(* PLC project Adressering.ecp, WAGO e!COCKPIT e!COCKPIT *)
(* stored: creationDateTime 2021-01-18T14:20:23.2110188, modificationDateTime 2021-01-18T11:51:27.6823754 *)

TYPE dtRomtype_1 : STRUCT
  RB601_V : BOOL;  (* Bevegelse *)
END_STRUCT;
END_TYPE

TYPE dtRomtype_11 : STRUCT
  RB601_V : BOOL;  (* Bevegelse *)
  RB601_HVAC : BOOL;  (* HVAC signal *)
END_STRUCT;
END_TYPE

TYPE dtRomtype_111 : STRUCT
  RB601_V : BOOL;  (* Bevegelse *)
  RB601_HVAC : BOOL;  (* HVAC signal *)
  RT601_CT : REAL;  (* Rom temperatur *)
  RT601_SP_D : REAL;  (* Temperatur SP *)
  RT601_SP_S : REAL;  (* Temperatur SP standby *)
  RT601_SP_N : REAL;  (* Temperatur SP nattsenk *)
  RT601_SP_F : REAL;  (* Temperatur SP frostsikring *)
  RT601_CS : REAL;  (* Aktivt temperatur SP *)
  OPM : REAL;  (* Rom modus *)
  OPM_CV : REAL;  (* Rom modus verdi *)
END_STRUCT;
END_TYPE

TYPE dtRomtype_1111 : STRUCT
  RB601_V : BOOL;  (* Bevegelse *)
  RB601_HVAC : BOOL;  (* HVAC signal *)
  RT601_CT : REAL;  (* Rom temperatur *)
  RT601_SP_D : REAL;  (* Temperatur SP *)
  RT601_SP_S : REAL;  (* Temperatur SP standby *)
  RT601_SP_N : REAL;  (* Temperatur SP nattsenk *)
  RT601_SP_F : REAL;  (* Temperatur SP frostsikring *)
  RT601_CS : REAL;  (* Aktivt temperatur SP *)
  OPM : REAL;  (* Rom modus *)
  OPM_CV : REAL;  (* Rom modus verdi *)
  RY601_CV : REAL;  (* Co2 Nivaa *)
  RY601_SP : REAL;  (* Co2 SP *)
  RY601_OP : REAL;  (* Co2 paadrag *)
END_STRUCT;
END_TYPE

TYPE dtRomtype_11101 : STRUCT
  RB601_V : BOOL;  (* Bevegelse *)
  RB601_HVAC : BOOL;  (* HVAC signal *)
  RT601_CT : REAL;  (* Rom temperatur *)
  RT601_SP_D : REAL;  (* Temperatur SP *)
  RT601_SP_S : REAL;  (* Temperatur SP standby *)
  RT601_SP_N : REAL;  (* Temperatur SP nattsenk *)
  RT601_SP_F : REAL;  (* Temperatur SP frostsikring *)
  RT601_CS : REAL;  (* Aktivt temperatur SP *)
  OPM : REAL;  (* Rom modus *)
  OPM_CV : REAL;  (* Rom modus verdi *)
  LH601_OP : REAL;  (* Varmepaadrag *)
  SB601_MAN : REAL;  (* Varmepaadrag force *)
END_STRUCT;
END_TYPE

TYPE dtRomtype_111011 : STRUCT
  RB601_V : BOOL;  (* Bevegelse *)
  RB601_HVAC : BOOL;  (* HVAC signal *)
  RT601_CT : REAL;  (* Rom temperatur *)
  RT601_SP_D : REAL;  (* Temperatur SP *)
  RT601_SP_S : REAL;  (* Temperatur SP standby *)
  RT601_SP_N : REAL;  (* Temperatur SP nattsenk *)
  RT601_SP_F : REAL;  (* Temperatur SP frostsikring *)
  RT601_CS : REAL;  (* Aktivt temperatur SP *)
  OPM : REAL;  (* Rom modus *)
  OPM_CV : REAL;  (* Rom modus verdi *)
  LH601_OP : REAL;  (* Varmepaadrag *)
  SB601_MAN : REAL;  (* Varmepaadrag force *)
  LH601_CMD : BOOL;  (* LH601_CMD *)
END_STRUCT;
END_TYPE

TYPE dtRomtype_1110111 : STRUCT
  RB601_V : BOOL;  (* Bevegelse *)
  RB601_HVAC : BOOL;  (* HVAC signal *)
  RT601_CT : REAL;  (* Rom temperatur *)
  RT601_SP_D : REAL;  (* Temperatur SP *)
  RT601_SP_S : REAL;  (* Temperatur SP standby *)
  RT601_SP_N : REAL;  (* Temperatur SP nattsenk *)
  RT601_SP_F : REAL;  (* Temperatur SP frostsikring *)
  RT601_CS : REAL;  (* Aktivt temperatur SP *)
  OPM : REAL;  (* Rom modus *)
  OPM_CV : REAL;  (* Rom modus verdi *)
  LH601_OP : REAL;  (* Varmepaadrag *)
  SB601_MAN : REAL;  (* Varmepaadrag force *)
  LH601_CMD : BOOL;  (* LH601_CMD *)
  LC601_OP : REAL;  (* LC601_OP *)
  LC601_MAN : REAL;  (* LC601 Force *)
END_STRUCT;
END_TYPE

TYPE dtRomtype_11111111 : STRUCT
  RB601_V : BOOL;  (* Bevegelse *)
  RB601_HVAC : BOOL;  (* HVAC signal *)
  RT601_CT : REAL;  (* Rom temperatur *)
  RT601_SP_D : REAL;  (* Temperatur SP *)
  RT601_SP_S : REAL;  (* Temperatur SP standby *)
  RT601_SP_N : REAL;  (* Temperatur SP nattsenk *)
  RT601_SP_F : REAL;  (* Temperatur SP frostsikring *)
  RT601_CS : REAL;  (* Aktivt temperatur SP *)
  OPM : REAL;  (* Rom modus *)
  OPM_CV : REAL;  (* Rom modus verdi *)
  RY601_CV : REAL;  (* Co2 Nivaa *)
  RY601_SP : REAL;  (* Co2 SP *)
  RY601_OP : REAL;  (* Co2 paadrag *)
  LH601_OP : REAL;  (* Varmepaadrag *)
  SB601_MAN : REAL;  (* Varmepaadrag force *)
  LH601_CMD : BOOL;  (* LH601_CMD *)
  LC601_OP : REAL;  (* LC601_OP *)
  LC601_MAN : REAL;  (* LC601 Force *)
  LC601_CMD : BOOL;  (* LC601_CMD *)
END_STRUCT;
END_TYPE

TYPE dtRomtype_111010111 : STRUCT
  RB601_V : BOOL;  (* Bevegelse *)
  RB601_HVAC : BOOL;  (* HVAC signal *)
  RT601_CT : REAL;  (* Rom temperatur *)
  RT601_SP_D : REAL;  (* Temperatur SP *)
  RT601_SP_S : REAL;  (* Temperatur SP standby *)
  RT601_SP_N : REAL;  (* Temperatur SP nattsenk *)
  RT601_SP_F : REAL;  (* Temperatur SP frostsikring *)
  RT601_CS : REAL;  (* Aktivt temperatur SP *)
  OPM : REAL;  (* Rom modus *)
  OPM_CV : REAL;  (* Rom modus verdi *)
  LH601_OP : REAL;  (* Varmepaadrag *)
  SB601_MAN : REAL;  (* Varmepaadrag force *)
  LC601_OP : REAL;  (* LC601_OP *)
  LC601_MAN : REAL;  (* LC601 Force *)
  LC601_CMD : BOOL;  (* LC601_CMD *)
  RT601_SP : REAL;  (* Temperatur SP feedback *)
END_STRUCT;
END_TYPE

TYPE dtRomtype_1111101011 : STRUCT
  RB601_V : BOOL;  (* Bevegelse *)
  RB601_HVAC : BOOL;  (* HVAC signal *)
  RT601_CT : REAL;  (* Rom temperatur *)
  RT601_SP_D : REAL;  (* Temperatur SP *)
  RT601_SP_S : REAL;  (* Temperatur SP standby *)
  RT601_SP_N : REAL;  (* Temperatur SP nattsenk *)
  RT601_SP_F : REAL;  (* Temperatur SP frostsikring *)
  RT601_CS : REAL;  (* Aktivt temperatur SP *)
  OPM : REAL;  (* Rom modus *)
  OPM_CV : REAL;  (* Rom modus verdi *)
  RY601_CV : REAL;  (* Co2 Nivaa *)
  RY601_SP : REAL;  (* Co2 SP *)
  RY601_OP : REAL;  (* Co2 paadrag *)
  LH601_OP : REAL;  (* Varmepaadrag *)
  SB601_MAN : REAL;  (* Varmepaadrag force *)
  LC601_OP : REAL;  (* LC601_OP *)
  LC601_MAN : REAL;  (* LC601 Force *)
  RT601_SP : REAL;  (* Temperatur SP feedback *)
  RT601_SP_FB : REAL;  (* Temperatur SP *)
  RT601_SP_IN : REAL;  (* Temperatur SP lokalt panel *)
END_STRUCT;
END_TYPE

TYPE dtRomtype_2111111111 : STRUCT
  RB601_V : BOOL;  (* Bevegelse *)
  RB602_V : BOOL;  (* Bevegelse *)
  RB601_HVAC : BOOL;  (* HVAC signal *)
  RT601_CT : REAL;  (* Rom temperatur *)
  RT601_SP_D : REAL;  (* Temperatur SP *)
  RT601_SP_S : REAL;  (* Temperatur SP standby *)
  RT601_SP_N : REAL;  (* Temperatur SP nattsenk *)
  RT601_SP_F : REAL;  (* Temperatur SP frostsikring *)
  RT601_CS : REAL;  (* Aktivt temperatur SP *)
  OPM : REAL;  (* Rom modus *)
  OPM_CV : REAL;  (* Rom modus verdi *)
  RY601_CV : REAL;  (* Co2 Nivaa *)
  RY601_SP : REAL;  (* Co2 SP *)
  RY601_OP : REAL;  (* Co2 paadrag *)
  LH601_OP : REAL;  (* Varmepaadrag *)
  SB601_MAN : REAL;  (* Varmepaadrag force *)
  LH601_CMD : BOOL;  (* LH601_CMD *)
  LC601_OP : REAL;  (* LC601_OP *)
  LC601_MAN : REAL;  (* LC601 Force *)
  LC601_CMD : BOOL;  (* LC601_CMD *)
  RT601_SP : REAL;  (* Temperatur SP feedback *)
  RT601_SP_FB : REAL;  (* Temperatur SP *)
  RT601_SP_IN : REAL;  (* Temperatur SP lokalt panel *)
END_STRUCT;
END_TYPE

TYPE dtRomtype_1211111111 : STRUCT
  RB601_V : BOOL;  (* Bevegelse *)
  RB601_HVAC : BOOL;  (* HVAC signal *)
  RB602_HVAC : BOOL;  (* HVAC signal *)
  RT601_CT : REAL;  (* Rom temperatur *)
  RT601_SP_D : REAL;  (* Temperatur SP *)
  RT601_SP_S : REAL;  (* Temperatur SP standby *)
  RT601_SP_N : REAL;  (* Temperatur SP nattsenk *)
  RT601_SP_F : REAL;  (* Temperatur SP frostsikring *)
  RT601_CS : REAL;  (* Aktivt temperatur SP *)
  OPM : REAL;  (* Rom modus *)
  OPM_CV : REAL;  (* Rom modus verdi *)
  RY601_CV : REAL;  (* Co2 Nivaa *)
  RY601_SP : REAL;  (* Co2 SP *)
  RY601_OP : REAL;  (* Co2 paadrag *)
  LH601_OP : REAL;  (* Varmepaadrag *)
  SB601_MAN : REAL;  (* Varmepaadrag force *)
  LH601_CMD : BOOL;  (* LH601_CMD *)
  LC601_OP : REAL;  (* LC601_OP *)
  LC601_MAN : REAL;  (* LC601 Force *)
  LC601_CMD : BOOL;  (* LC601_CMD *)
  RT601_SP : REAL;  (* Temperatur SP feedback *)
  RT601_SP_FB : REAL;  (* Temperatur SP *)
  RT601_SP_IN : REAL;  (* Temperatur SP lokalt panel *)
END_STRUCT;
END_TYPE

TYPE dtRomtype_1121111111 : STRUCT
  RB601_V : BOOL;  (* Bevegelse *)
  RB601_HVAC : BOOL;  (* HVAC signal *)
  RT601_CT : REAL;  (* Rom temperatur *)
  RT602_CT : REAL;  (* Rom temperatur *)
  RT601_SP_D : REAL;  (* Temperatur SP *)
  RT601_SP_S : REAL;  (* Temperatur SP standby *)
  RT601_SP_N : REAL;  (* Temperatur SP nattsenk *)
  RT601_SP_F : REAL;  (* Temperatur SP frostsikring *)
  RT601_CS : REAL;  (* Aktivt temperatur SP *)
  OPM : REAL;  (* Rom modus *)
  OPM_CV : REAL;  (* Rom modus verdi *)
  RY601_CV : REAL;  (* Co2 Nivaa *)
  RY601_SP : REAL;  (* Co2 SP *)
  RY601_OP : REAL;  (* Co2 paadrag *)
  LH601_OP : REAL;  (* Varmepaadrag *)
  SB601_MAN : REAL;  (* Varmepaadrag force *)
  LH601_CMD : BOOL;  (* LH601_CMD *)
  LC601_OP : REAL;  (* LC601_OP *)
  LC601_MAN : REAL;  (* LC601 Force *)
  LC601_CMD : BOOL;  (* LC601_CMD *)
  RT601_SP : REAL;  (* Temperatur SP feedback *)
  RT601_SP_FB : REAL;  (* Temperatur SP *)
  RT601_SP_IN : REAL;  (* Temperatur SP lokalt panel *)
END_STRUCT;
END_TYPE

TYPE dtRomtype_1112111111 : STRUCT
  RB601_V : BOOL;  (* Bevegelse *)
  RB601_HVAC : BOOL;  (* HVAC signal *)
  RT601_CT : REAL;  (* Rom temperatur *)
  RT601_SP_D : REAL;  (* Temperatur SP *)
  RT601_SP_S : REAL;  (* Temperatur SP standby *)
  RT601_SP_N : REAL;  (* Temperatur SP nattsenk *)
  RT601_SP_F : REAL;  (* Temperatur SP frostsikring *)
  RT601_CS : REAL;  (* Aktivt temperatur SP *)
  OPM : REAL;  (* Rom modus *)
  OPM_CV : REAL;  (* Rom modus verdi *)
  RY601_CV : REAL;  (* Co2 Nivaa *)
  RY601_SP : REAL;  (* Co2 SP *)
  RY601_OP : REAL;  (* Co2 paadrag *)
  RY602_CV : REAL;  (* Co2 Nivaa *)
  RY602_SP : REAL;  (* Co2 SP *)
  RY602_OP : REAL;  (* Co2 paadrag *)
  LH601_OP : REAL;  (* Varmepaadrag *)
  SB601_MAN : REAL;  (* Varmepaadrag force *)
  LH601_CMD : BOOL;  (* LH601_CMD *)
  LC601_OP : REAL;  (* LC601_OP *)
  LC601_MAN : REAL;  (* LC601 Force *)
  LC601_CMD : BOOL;  (* LC601_CMD *)
  RT601_SP : REAL;  (* Temperatur SP feedback *)
  RT601_SP_FB : REAL;  (* Temperatur SP *)
  RT601_SP_IN : REAL;  (* Temperatur SP lokalt panel *)
END_STRUCT;
END_TYPE

TYPE dtRomtype_1111211111 : STRUCT
  RB601_V : BOOL;  (* Bevegelse *)
  RB601_HVAC : BOOL;  (* HVAC signal *)
  RT601_CT : REAL;  (* Rom temperatur *)
  RT601_SP_D : REAL;  (* Temperatur SP *)
  RT601_SP_S : REAL;  (* Temperatur SP standby *)
  RT601_SP_N : REAL;  (* Temperatur SP nattsenk *)
  RT601_SP_F : REAL;  (* Temperatur SP frostsikring *)
  RT601_CS : REAL;  (* Aktivt temperatur SP *)
  OPM : REAL;  (* Rom modus *)
  OPM_CV : REAL;  (* Rom modus verdi *)
  RY601_CV : REAL;  (* Co2 Nivaa *)
  RY601_SP : REAL;  (* Co2 SP *)
  RY601_OP : REAL;  (* Co2 paadrag *)
  LH601_OP : REAL;  (* Varmepaadrag *)
  LH602_OP : REAL;  (* Varmepaadrag *)
  SB601_MAN : REAL;  (* Varmepaadrag force *)
  LH601_CMD : BOOL;  (* LH601_CMD *)
  LC601_OP : REAL;  (* LC601_OP *)
  LC601_MAN : REAL;  (* LC601 Force *)
  LC601_CMD : BOOL;  (* LC601_CMD *)
  RT601_SP : REAL;  (* Temperatur SP feedback *)
  RT601_SP_FB : REAL;  (* Temperatur SP *)
  RT601_SP_IN : REAL;  (* Temperatur SP lokalt panel *)
END_STRUCT;
END_TYPE

TYPE dtRomtype_1111112111 : STRUCT
  RB601_V : BOOL;  (* Bevegelse *)
  RB601_HVAC : BOOL;  (* HVAC signal *)
  RT601_CT : REAL;  (* Rom temperatur *)
  RT601_SP_D : REAL;  (* Temperatur SP *)
  RT601_SP_S : REAL;  (* Temperatur SP standby *)
  RT601_SP_N : REAL;  (* Temperatur SP nattsenk *)
  RT601_SP_F : REAL;  (* Temperatur SP frostsikring *)
  RT601_CS : REAL;  (* Aktivt temperatur SP *)
  OPM : REAL;  (* Rom modus *)
  OPM_CV : REAL;  (* Rom modus verdi *)
  RY601_CV : REAL;  (* Co2 Nivaa *)
  RY601_SP : REAL;  (* Co2 SP *)
  RY601_OP : REAL;  (* Co2 paadrag *)
  LH601_OP : REAL;  (* Varmepaadrag *)
  SB601_MAN : REAL;  (* Varmepaadrag force *)
  LH601_CMD : BOOL;  (* LH601_CMD *)
  LC601_OP : REAL;  (* LC601_OP *)
  LC602_OP : REAL;  (* LC602_OP *)
  LC601_MAN : REAL;  (* LC601 Force *)
  LC601_CMD : BOOL;  (* LC601_CMD *)
  RT601_SP : REAL;  (* Temperatur SP feedback *)
  RT601_SP_FB : REAL;  (* Temperatur SP *)
  RT601_SP_IN : REAL;  (* Temperatur SP lokalt panel *)
END_STRUCT;
END_TYPE

TYPE dtRomtype_1111111211 : STRUCT
  RB601_V : BOOL;  (* Bevegelse *)
  RB601_HVAC : BOOL;  (* HVAC signal *)
  RT601_CT : REAL;  (* Rom temperatur *)
  RT601_SP_D : REAL;  (* Temperatur SP *)
  RT601_SP_S : REAL;  (* Temperatur SP standby *)
  RT601_SP_N : REAL;  (* Temperatur SP nattsenk *)
  RT601_SP_F : REAL;  (* Temperatur SP frostsikring *)
  RT601_CS : REAL;  (* Aktivt temperatur SP *)
  OPM : REAL;  (* Rom modus *)
  OPM_CV : REAL;  (* Rom modus verdi *)
  RY601_CV : REAL;  (* Co2 Nivaa *)
  RY601_SP : REAL;  (* Co2 SP *)
  RY601_OP : REAL;  (* Co2 paadrag *)
  LH601_OP : REAL;  (* Varmepaadrag *)
  SB601_MAN : REAL;  (* Varmepaadrag force *)
  LH601_CMD : BOOL;  (* LH601_CMD *)
  LC601_OP : REAL;  (* LC601_OP *)
  LC601_MAN : REAL;  (* LC601 Force *)
  LC601_CMD : BOOL;  (* LC601_CMD *)
  LC602_CMD : BOOL;  (* LC602_CMD *)
  RT601_SP : REAL;  (* Temperatur SP feedback *)
  RT601_SP_FB : REAL;  (* Temperatur SP *)
  RT601_SP_IN : REAL;  (* Temperatur SP lokalt panel *)
END_STRUCT;
END_TYPE

TYPE dtRomtype_1121111121 : STRUCT
  RB601_V : BOOL;  (* Bevegelse *)
  RB601_HVAC : BOOL;  (* HVAC signal *)
  RT601_CT : REAL;  (* Rom temperatur *)
  RT602_CT : REAL;  (* Rom temperatur *)
  RT601_SP_D : REAL;  (* Temperatur SP *)
  RT601_SP_S : REAL;  (* Temperatur SP standby *)
  RT601_SP_N : REAL;  (* Temperatur SP nattsenk *)
  RT601_SP_F : REAL;  (* Temperatur SP frostsikring *)
  RT601_CS : REAL;  (* Aktivt temperatur SP *)
  OPM : REAL;  (* Rom modus *)
  OPM_CV : REAL;  (* Rom modus verdi *)
  RY601_CV : REAL;  (* Co2 Nivaa *)
  RY601_SP : REAL;  (* Co2 SP *)
  RY601_OP : REAL;  (* Co2 paadrag *)
  LH601_OP : REAL;  (* Varmepaadrag *)
  SB601_MAN : REAL;  (* Varmepaadrag force *)
  LH601_CMD : BOOL;  (* LH601_CMD *)
  LC601_OP : REAL;  (* LC601_OP *)
  LC601_MAN : REAL;  (* LC601 Force *)
  LC601_CMD : BOOL;  (* LC601_CMD *)
  RT601_SP : REAL;  (* Temperatur SP feedback *)
  RT601_SP_FB : REAL;  (* Temperatur SP *)
  RT601_SP_IN : REAL;  (* Temperatur SP lokalt panel *)
END_STRUCT;
END_TYPE

TYPE dtRomtype_1111111112 : STRUCT
  RB601_V : BOOL;  (* Bevegelse *)
  RB601_HVAC : BOOL;  (* HVAC signal *)
  RT601_CT : REAL;  (* Rom temperatur *)
  RT601_SP_D : REAL;  (* Temperatur SP *)
  RT601_SP_S : REAL;  (* Temperatur SP standby *)
  RT601_SP_N : REAL;  (* Temperatur SP nattsenk *)
  RT601_SP_F : REAL;  (* Temperatur SP frostsikring *)
  RT601_CS : REAL;  (* Aktivt temperatur SP *)
  OPM : REAL;  (* Rom modus *)
  OPM_CV : REAL;  (* Rom modus verdi *)
  RY601_CV : REAL;  (* Co2 Nivaa *)
  RY601_SP : REAL;  (* Co2 SP *)
  RY601_OP : REAL;  (* Co2 paadrag *)
  LH601_OP : REAL;  (* Varmepaadrag *)
  SB601_MAN : REAL;  (* Varmepaadrag force *)
  LH601_CMD : BOOL;  (* LH601_CMD *)
  LC601_OP : REAL;  (* LC601_OP *)
  LC601_MAN : REAL;  (* LC601 Force *)
  LC601_CMD : BOOL;  (* LC601_CMD *)
  RT601_SP : REAL;  (* Temperatur SP feedback *)
  RT601_SP_FB : REAL;  (* Temperatur SP *)
  RT601_SP_IN : REAL;  (* Temperatur SP lokalt panel *)
  RT602_SP_FB : REAL;  (* Temperatur SP *)
  RT602_SP_IN : REAL;  (* Temperatur SP lokalt panel *)
END_STRUCT;
END_TYPE

TYPE dtRomtype_4111111111 : STRUCT
  RB601_V : BOOL;  (* Bevegelse *)
  RB602_V : BOOL;  (* Bevegelse *)
  RB603_V : BOOL;  (* Bevegelse *)
  RB604_V : BOOL;  (* Bevegelse *)
  RB601_HVAC : BOOL;  (* HVAC signal *)
  RT601_CT : REAL;  (* Rom temperatur *)
  RT601_SP_D : REAL;  (* Temperatur SP *)
  RT601_SP_S : REAL;  (* Temperatur SP standby *)
  RT601_SP_N : REAL;  (* Temperatur SP nattsenk *)
  RT601_SP_F : REAL;  (* Temperatur SP frostsikring *)
  RT601_CS : REAL;  (* Aktivt temperatur SP *)
  OPM : REAL;  (* Rom modus *)
  OPM_CV : REAL;  (* Rom modus verdi *)
  RY601_CV : REAL;  (* Co2 Nivaa *)
  RY601_SP : REAL;  (* Co2 SP *)
  RY601_OP : REAL;  (* Co2 paadrag *)
  LH601_OP : REAL;  (* Varmepaadrag *)
  SB601_MAN : REAL;  (* Varmepaadrag force *)
  LH601_CMD : BOOL;  (* LH601_CMD *)
  LC601_OP : REAL;  (* LC601_OP *)
  LC601_MAN : REAL;  (* LC601 Force *)
  LC601_CMD : BOOL;  (* LC601_CMD *)
  RT601_SP : REAL;  (* Temperatur SP feedback *)
  RT601_SP_FB : REAL;  (* Temperatur SP *)
  RT601_SP_IN : REAL;  (* Temperatur SP lokalt panel *)
END_STRUCT;
END_TYPE

TYPE dtRomtype_5521111111 : STRUCT
  RB601_V : BOOL;  (* Bevegelse *)
  RB602_V : BOOL;  (* Bevegelse *)
  RB603_V : BOOL;  (* Bevegelse *)
  RB604_V : BOOL;  (* Bevegelse *)
  RB605_V : BOOL;  (* Bevegelse *)
  RB601_HVAC : BOOL;  (* HVAC signal *)
  RB602_HVAC : BOOL;  (* HVAC signal *)
  RB603_HVAC : BOOL;  (* HVAC signal *)
  RB604_HVAC : BOOL;  (* HVAC signal *)
  RB605_HVAC : BOOL;  (* HVAC signal *)
  RT601_CT : REAL;  (* Rom temperatur *)
  RT602_CT : REAL;  (* Rom temperatur *)
  RT601_SP_D : REAL;  (* Temperatur SP *)
  RT601_SP_S : REAL;  (* Temperatur SP standby *)
  RT601_SP_N : REAL;  (* Temperatur SP nattsenk *)
  RT601_SP_F : REAL;  (* Temperatur SP frostsikring *)
  RT601_CS : REAL;  (* Aktivt temperatur SP *)
  OPM : REAL;  (* Rom modus *)
  OPM_CV : REAL;  (* Rom modus verdi *)
  RY601_CV : REAL;  (* Co2 Nivaa *)
  RY601_SP : REAL;  (* Co2 SP *)
  RY601_OP : REAL;  (* Co2 paadrag *)
  LH601_OP : REAL;  (* Varmepaadrag *)
  SB601_MAN : REAL;  (* Varmepaadrag force *)
  LH601_CMD : BOOL;  (* LH601_CMD *)
  LC601_OP : REAL;  (* LC601_OP *)
  LC601_MAN : REAL;  (* LC601 Force *)
  LC601_CMD : BOOL;  (* LC601_CMD *)
  RT601_SP : REAL;  (* Temperatur SP feedback *)
  RT601_SP_FB : REAL;  (* Temperatur SP *)
  RT601_SP_IN : REAL;  (* Temperatur SP lokalt panel *)
END_STRUCT;
END_TYPE

TYPE dtRomtype_1111111111 : STRUCT
  RB601_V : BOOL;  (* Bevegelse *)
  RB601_HVAC : BOOL;  (* HVAC signal *)
  RT601_CT : REAL;  (* Rom temperatur *)
  RT601_SP_D : REAL;  (* Temperatur SP *)
  RT601_SP_S : REAL;  (* Temperatur SP standby *)
  RT601_SP_N : REAL;  (* Temperatur SP nattsenk *)
  RT601_SP_F : REAL;  (* Temperatur SP frostsikring *)
  RT601_CS : REAL;  (* Aktivt temperatur SP *)
  OPM : REAL;  (* Rom modus *)
  OPM_CV : REAL;  (* Rom modus verdi *)
  RY601_CV : REAL;  (* Co2 Nivaa *)
  RY601_SP : REAL;  (* Co2 SP *)
  RY601_OP : REAL;  (* Co2 paadrag *)
  LH601_OP : REAL;  (* Varmepaadrag *)
  SB601_MAN : REAL;  (* Varmepaadrag force *)
  LH601_CMD : BOOL;  (* LH601_CMD *)
  LC601_OP : REAL;  (* LC601_OP *)
  LC601_MAN : REAL;  (* LC601 Force *)
  LC601_CMD : BOOL;  (* LC601_CMD *)
  RT601_SP : REAL;  (* Temperatur SP feedback *)
  RT601_SP_FB : REAL;  (* Temperatur SP *)
  RT601_SP_IN : REAL;  (* Temperatur SP lokalt panel *)
END_STRUCT;
END_TYPE

{attribute 'qualified_only'}
VAR_GLOBAL  (* STLV80_563 *)
  STLV80_A_563_KNX_Card_1_Status : BOOL;  (* KNX kort 1 status *)
  STLV80_A_563_KNX_Card_2_Status : BOOL;  (* KNX kort 2 status *)
  STLV80_A_563_KNX_Card_3_Status : BOOL;  (* KNX kort 3 status *)
  STLV80_A_563_5A201 : dtRomtype_1;  (* rom1 *)
  STLV80_A_563_5A202 : dtRomtype_11;  (* rom1 *)
  STLV80_A_563_5A301 : dtRomtype_111;  (* rom1 *)
  STLV80_A_563_5A302 : dtRomtype_1111;  (* rom1 *)
  STLV80_A_563_5B201 : dtRomtype_11101;  (* rom1 *)
  STLV80_A_563_5B202 : dtRomtype_111011;  (* rom1 *)
  STLV80_A_563_5B301 : dtRomtype_1110111;  (* rom1 *)
  STLV80_A_563_5B302 : dtRomtype_11111111;  (* rom1 *)
  STLV80_A_563_5C201 : dtRomtype_111010111;  (* rom1 *)
  STLV80_A_563_5C202 : dtRomtype_1111101011;  (* rom1 *)
  STLV80_A_563_5C301 : dtRomtype_11111111;  (* rom1 *)
  STLV80_A_563_5C302 : dtRomtype_2111111111;  (* rom1 *)
  STLV80_A_563_5D201 : dtRomtype_1211111111;  (* rom1 *)
  STLV80_A_563_5D202 : dtRomtype_1121111111;  (* rom1 *)
  STLV80_A_563_5D301 : dtRomtype_1112111111;  (* rom1 *)
  STLV80_A_563_5D302 : dtRomtype_1111211111;  (* rom1 *)
  STLV80_A_563_5E201 : dtRomtype_1111112111;  (* rom1 *)
  STLV80_A_563_5E202 : dtRomtype_1111111211;  (* rom1 *)
  STLV80_A_563_5E301 : dtRomtype_1121111121;  (* rom1 *)
  STLV80_A_563_5E302 : dtRomtype_1111111112;  (* rom1 *)
  STLV80_A_563_5F201 : dtRomtype_4111111111;  (* rom1 *)
  STLV80_A_563_5F202 : dtRomtype_5521111111;  (* rom1 *)
  STLV80_A_563_5F301 : dtRomtype_1111111111;  (* rom1 *)
  STLV80_A_563_5F302 : dtRomtype_1111111111;  (* rom1 *)
  STLV80_A_563_5G201 : dtRomtype_1111111111;  (* rom1 *)
  STLV80_A_563_5G202 : dtRomtype_1111111111;  (* rom1 *)
  STLV80_A_563_5H301 : dtRomtype_1111111111;  (* rom1 *)
  STLV80_A_563_5H302 : dtRomtype_1111111111;  (* rom1 *)
  STLV80_A_563_5H201 : dtRomtype_1111111111;  (* rom1 *)
  STLV80_A_563_5I202 : dtRomtype_1111111111;  (* rom1 *)
  STLV80_A_563_5I301 : dtRomtype_1111111111;  (* rom1 *)
  STLV80_A_563_5I302 : dtRomtype_1111111111;  (* rom1 *)
  STLV80_A_563_5J201 : dtRomtype_1111111111;  (* rom1 *)
  STLV80_A_563_5J202 : dtRomtype_1111111111;  (* rom1 *)
  STLV80_A_563_5J301 : dtRomtype_1111111111;  (* rom1 *)
  STLV80_A_563_5K302 : dtRomtype_1111111111;  (* rom1 *)
  STLV80_A_563_5K201 : dtRomtype_1111111111;  (* rom1 *)
  STLV80_A_563_5K202 : dtRomtype_1111111111;  (* rom1 *)
  STLV80_A_563_5K301 : dtRomtype_1111111111;  (* rom1 *)
  STLV80_A_563_5L201 : dtRomtype_1111111111;  (* rom1 *)
  STLV80_A_563_5L202 : dtRomtype_1111111111;  (* rom1 *)
  STLV80_A_563_5L301 : dtRomtype_1111111111;  (* rom1 *)
  STLV80_A_563_5L302 : dtRomtype_1111111111;  (* rom1 *)
  STLV80_A_563_5M201 : dtRomtype_1111111111;  (* rom1 *)
  STLV80_A_563_5M202 : dtRomtype_1111111111;  (* rom1 *)
  STLV80_A_563_5M301 : dtRomtype_1111111111;  (* rom1 *)
  STLV80_A_563_5N201 : dtRomtype_1111111111;  (* rom1 *)
  STLV80_A_563_5N202 : dtRomtype_1111111111;  (* rom1 *)
  STLV80_A_563_5N301 : dtRomtype_1111111111;  (* rom1 *)
  STLV80_A_563_5N302 : dtRomtype_1111111111;  (* rom1 *)
  STLV80_A_563_5O302 : dtRomtype_1111111111;  (* rom1 *)
  STLV80_A_563_5O201 : dtRomtype_1111111111;  (* rom1 *)
  STLV80_A_563_5O202 : dtRomtype_1111111111;  (* rom1 *)
  STLV80_A_563_5O301 : dtRomtype_1111111111;  (* rom1 *)
  STLV80_A_563_5P302 : dtRomtype_1111111111;  (* rom1 *)
  STLV80_A_563_5P201 : dtRomtype_1111111111;  (* rom1 *)
  STLV80_A_563_5P202 : dtRomtype_1111111111;  (* rom1 *)
  STLV80_A_563_5Q301 : dtRomtype_1111111111;  (* rom1 *)
  STLV80_A_563_5Q302 : dtRomtype_1111111111;  (* rom1 *)
END_VAR

PROGRAM PRG_563_KNX_1
  VAR
    i : INT := 0;  (* Felles *)
    Interval : OSCAT_BASIC.CLK_PRG;
    typDPT : typDPT;
    KNX_master_1 : WagoAppKNX.FbKNX_Master;  (* Master *)
    M1_001_5A201_RB601_V : fbDPT_Switch_pro;  (* 5A201 *)
    M1_002_5A202_RB601_V : fbDPT_Switch_pro;  (* 5A202 *)
    M1_003_5A202_RB601_HVAC : fbDPT_Switch_pro;
    M1_004_5A301_RB601_V : fbDPT_Switch_pro;  (* 5A301 *)
    M1_005_5A301_RB601_HVAC : fbDPT_Switch_pro;
    M1_006_5A301_RT601_CT : fbDPT_Value_Temp_pro;
    M1_007_5A302_RB601_V : fbDPT_Switch_pro;  (* 5A302 *)
    M1_008_5A302_RB601_HVAC : fbDPT_Switch_pro;
    M1_009_5A302_RT601_CT : fbDPT_Value_Temp_pro;
    M1_010_5A302_RY601_CV : fbDPT_Value_AirQuality_pro;
    M1_011_5B201_RB601_V : fbDPT_Switch_pro;  (* 5B201 *)
    M1_012_5B201_RB601_HVAC : fbDPT_Switch_pro;
    M1_013_5B201_RT601_CT : fbDPT_Value_Temp_pro;
    M1_014_5B201_LH601_OP : fbDPT_Scaling_pro;
    M1_015_5B202_RB601_V : fbDPT_Switch_pro;  (* 5B202 *)
    M1_016_5B202_RB601_HVAC : fbDPT_Switch_pro;
    M1_017_5B202_RT601_CT : fbDPT_Value_Temp_pro;
    M1_018_5B202_LH601_OP : fbDPT_Scaling_pro;
    M1_019_5B202_LH601_CMD : fbDPT_Switch_pro;
    M1_020_5B301_RB601_V : fbDPT_Switch_pro;  (* 5B301 *)
    M1_021_5B301_RB601_HVAC : fbDPT_Switch_pro;
    M1_022_5B301_RT601_CT : fbDPT_Value_Temp_pro;
    M1_023_5B301_LH601_OP : fbDPT_Scaling_pro;
    M1_024_5B301_LH601_CMD : fbDPT_Switch_pro;
    M1_025_5B301_LC601_OP : fbDPT_Scaling_pro;
    M1_026_5B302_RB601_V : fbDPT_Switch_pro;  (* 5B302 *)
    M1_027_5B302_RB601_HVAC : fbDPT_Switch_pro;
    M1_028_5B302_RT601_CT : fbDPT_Value_Temp_pro;
    M1_029_5B302_RY601_CV : fbDPT_Value_AirQuality_pro;
    M1_030_5B302_LH601_OP : fbDPT_Scaling_pro;
    M1_031_5B302_LH601_CMD : fbDPT_Switch_pro;
    M1_032_5B302_LC601_OP : fbDPT_Scaling_pro;
    M1_033_5B302_LC601_CMD : fbDPT_Switch_pro;
    M1_034_5C201_RB601_V : fbDPT_Switch_pro;  (* 5C201 *)
    M1_035_5C201_RB601_HVAC : fbDPT_Switch_pro;
    M1_036_5C201_RT601_CT : fbDPT_Value_Temp_pro;
    M1_037_5C201_LH601_OP : fbDPT_Scaling_pro;
    M1_038_5C201_LC601_OP : fbDPT_Scaling_pro;
    M1_039_5C201_LC601_CMD : fbDPT_Switch_pro;
    M1_040_5C201_RT601_SP : fbDPT_Value_Temp_pro;
    M1_041_5C202_RB601_V : fbDPT_Switch_pro;  (* 5C202 *)
    M1_042_5C202_RB601_HVAC : fbDPT_Switch_pro;
    M1_043_5C202_RT601_CT : fbDPT_Value_Temp_pro;
    M1_044_5C202_RY601_CV : fbDPT_Value_AirQuality_pro;
    M1_045_5C202_LH601_OP : fbDPT_Scaling_pro;
    M1_046_5C202_LC601_OP : fbDPT_Scaling_pro;
    M1_047_5C202_RT601_SP : fbDPT_Value_Temp_pro;
    M1_048_5C202_RT601_SP_FB : fbDPT_Value_Temp_pro;
    M1_049_5C301_RB601_V : fbDPT_Switch_pro;  (* 5C301 *)
    M1_050_5C301_RB601_HVAC : fbDPT_Switch_pro;
    M1_051_5C301_RT601_CT : fbDPT_Value_Temp_pro;
    M1_052_5C301_RY601_CV : fbDPT_Value_AirQuality_pro;
    M1_053_5C301_LH601_OP : fbDPT_Scaling_pro;
    M1_054_5C301_LH601_CMD : fbDPT_Switch_pro;
    M1_055_5C301_LC601_OP : fbDPT_Scaling_pro;
    M1_056_5C301_LC601_CMD : fbDPT_Switch_pro;
    M1_057_5C302_RB601_V : fbDPT_Switch_pro;  (* 5C302 *)
    M1_058_5C302_RB602_V : fbDPT_Switch_pro;
    M1_059_5C302_RB601_HVAC : fbDPT_Switch_pro;
    M1_060_5C302_RT601_CT : fbDPT_Value_Temp_pro;
    M1_061_5C302_RY601_CV : fbDPT_Value_AirQuality_pro;
    M1_062_5C302_LH601_OP : fbDPT_Scaling_pro;
    M1_063_5C302_LH601_CMD : fbDPT_Switch_pro;
    M1_064_5C302_LC601_OP : fbDPT_Scaling_pro;
    M1_065_5C302_LC601_CMD : fbDPT_Switch_pro;
    M1_066_5C302_RT601_SP : fbDPT_Value_Temp_pro;
    M1_067_5C302_RT601_SP_FB : fbDPT_Value_Temp_pro;
    M1_068_5D201_RB601_V : fbDPT_Switch_pro;  (* 5D201 *)
    M1_069_5D201_RB601_HVAC : fbDPT_Switch_pro;
    M1_070_5D201_RB602_HVAC : fbDPT_Switch_pro;
    M1_071_5D201_RT601_CT : fbDPT_Value_Temp_pro;
    M1_072_5D201_RY601_CV : fbDPT_Value_AirQuality_pro;
    M1_073_5D201_LH601_OP : fbDPT_Scaling_pro;
    M1_074_5D201_LH601_CMD : fbDPT_Switch_pro;
    M1_075_5D201_LC601_OP : fbDPT_Scaling_pro;
    M1_076_5D201_LC601_CMD : fbDPT_Switch_pro;
    M1_077_5D201_RT601_SP : fbDPT_Value_Temp_pro;
    M1_078_5D201_RT601_SP_FB : fbDPT_Value_Temp_pro;
    M1_079_5D202_RB601_V : fbDPT_Switch_pro;  (* 5D202 *)
    M1_080_5D202_RB601_HVAC : fbDPT_Switch_pro;
    M1_081_5D202_RT601_CT : fbDPT_Value_Temp_pro;
    M1_082_5D202_RT602_CT : fbDPT_Value_Temp_pro;
    M1_083_5D202_RY601_CV : fbDPT_Value_AirQuality_pro;
    M1_084_5D202_LH601_OP : fbDPT_Scaling_pro;
    M1_085_5D202_LH601_CMD : fbDPT_Switch_pro;
    M1_086_5D202_LC601_OP : fbDPT_Scaling_pro;
    M1_087_5D202_LC601_CMD : fbDPT_Switch_pro;
    M1_088_5D202_RT601_SP : fbDPT_Value_Temp_pro;
    M1_089_5D202_RT601_SP_FB : fbDPT_Value_Temp_pro;
    M1_090_5D301_RB601_V : fbDPT_Switch_pro;  (* 5D301 *)
    M1_091_5D301_RB601_HVAC : fbDPT_Switch_pro;
    M1_092_5D301_RT601_CT : fbDPT_Value_Temp_pro;
    M1_093_5D301_RY601_CV : fbDPT_Value_AirQuality_pro;
    M1_094_5D301_RY602_CV : fbDPT_Value_AirQuality_pro;
    M1_095_5D301_LH601_OP : fbDPT_Scaling_pro;
    M1_096_5D301_LH601_CMD : fbDPT_Switch_pro;
    M1_097_5D301_LC601_OP : fbDPT_Scaling_pro;
    M1_098_5D301_LC601_CMD : fbDPT_Switch_pro;
    M1_099_5D301_RT601_SP : fbDPT_Value_Temp_pro;
    M1_100_5D301_RT601_SP_FB : fbDPT_Value_Temp_pro;
    M1_101_5D302_RB601_V : fbDPT_Switch_pro;  (* 5D302 *)
    M1_102_5D302_RB601_HVAC : fbDPT_Switch_pro;
    M1_103_5D302_RT601_CT : fbDPT_Value_Temp_pro;
    M1_104_5D302_RY601_CV : fbDPT_Value_AirQuality_pro;
    M1_105_5D302_LH601_OP : fbDPT_Scaling_pro;
    M1_106_5D302_LH602_OP : fbDPT_Scaling_pro;
    M1_107_5D302_LH601_CMD : fbDPT_Switch_pro;
    M1_108_5D302_LC601_OP : fbDPT_Scaling_pro;
    M1_109_5D302_LC601_CMD : fbDPT_Switch_pro;
    M1_110_5D302_RT601_SP : fbDPT_Value_Temp_pro;
    M1_111_5D302_RT601_SP_FB : fbDPT_Value_Temp_pro;
    M1_112_5E201_RB601_V : fbDPT_Switch_pro;  (* 5E201 *)
    M1_113_5E201_RB601_HVAC : fbDPT_Switch_pro;
    M1_114_5E201_RT601_CT : fbDPT_Value_Temp_pro;
    M1_115_5E201_RY601_CV : fbDPT_Value_AirQuality_pro;
    M1_116_5E201_LH601_OP : fbDPT_Scaling_pro;
    M1_117_5E201_LH601_CMD : fbDPT_Switch_pro;
    M1_118_5E201_LC601_OP : fbDPT_Scaling_pro;
    M1_119_5E201_LC602_OP : fbDPT_Scaling_pro;
    M1_120_5E201_LC601_CMD : fbDPT_Switch_pro;
    M1_121_5E201_RT601_SP : fbDPT_Value_Temp_pro;
    M1_122_5E201_RT601_SP_FB : fbDPT_Value_Temp_pro;
    M1_123_5E202_RB601_V : fbDPT_Switch_pro;  (* 5E202 *)
    M1_124_5E202_RB601_HVAC : fbDPT_Switch_pro;
    M1_125_5E202_RT601_CT : fbDPT_Value_Temp_pro;
    M1_126_5E202_RY601_CV : fbDPT_Value_AirQuality_pro;
    M1_127_5E202_LH601_OP : fbDPT_Scaling_pro;
    M1_128_5E202_LH601_CMD : fbDPT_Switch_pro;
    M1_129_5E202_LC601_OP : fbDPT_Scaling_pro;
    M1_130_5E202_LC601_CMD : fbDPT_Switch_pro;
    M1_131_5E202_LC602_CMD : fbDPT_Switch_pro;
    M1_132_5E202_RT601_SP : fbDPT_Value_Temp_pro;
    M1_133_5E202_RT601_SP_FB : fbDPT_Value_Temp_pro;
    M1_134_5E301_RB601_V : fbDPT_Switch_pro;  (* 5E301 *)
    M1_135_5E301_RB601_HVAC : fbDPT_Switch_pro;
    M1_136_5E301_RT601_CT : fbDPT_Value_Temp_pro;
    M1_137_5E301_RT602_CT : fbDPT_Value_Temp_pro;
    M1_138_5E301_RY601_CV : fbDPT_Value_AirQuality_pro;
    M1_139_5E301_LH601_OP : fbDPT_Scaling_pro;
    M1_140_5E301_LH601_CMD : fbDPT_Switch_pro;
    M1_141_5E301_LC601_OP : fbDPT_Scaling_pro;
    M1_142_5E301_LC601_CMD : fbDPT_Switch_pro;
    M1_143_5E301_RT601_SP : fbDPT_Value_Temp_pro;
    M1_144_5E301_RT602_SP : fbDPT_Value_Temp_pro;
    M1_145_5E301_RT601_SP_FB : fbDPT_Value_Temp_pro;
    M1_146_5E302_RB601_V : fbDPT_Switch_pro;  (* 5E302 *)
    M1_147_5E302_RB601_HVAC : fbDPT_Switch_pro;
    M1_148_5E302_RT601_CT : fbDPT_Value_Temp_pro;
    M1_149_5E302_RY601_CV : fbDPT_Value_AirQuality_pro;
    M1_150_5E302_LH601_OP : fbDPT_Scaling_pro;
    M1_151_5E302_LH601_CMD : fbDPT_Switch_pro;
    M1_152_5E302_LC601_OP : fbDPT_Scaling_pro;
    M1_153_5E302_LC601_CMD : fbDPT_Switch_pro;
    M1_154_5E302_RT601_SP : fbDPT_Value_Temp_pro;
    M1_155_5E302_RT601_SP_FB : fbDPT_Value_Temp_pro;
    M1_156_5E302_RT602_SP_FB : fbDPT_Value_Temp_pro;
    M1_157_5F201_RB601_V : fbDPT_Switch_pro;  (* 5F201 *)
    M1_158_5F201_RB602_V : fbDPT_Switch_pro;
    M1_159_5F201_RB603_V : fbDPT_Switch_pro;
    M1_160_5F201_RB604_V : fbDPT_Switch_pro;
    M1_161_5F201_RB601_HVAC : fbDPT_Switch_pro;
    M1_162_5F201_RT601_CT : fbDPT_Value_Temp_pro;
    M1_163_5F201_RY601_CV : fbDPT_Value_AirQuality_pro;
    M1_164_5F201_LH601_OP : fbDPT_Scaling_pro;
    M1_165_5F201_LH601_CMD : fbDPT_Switch_pro;
    M1_166_5F201_LC601_OP : fbDPT_Scaling_pro;
    M1_167_5F201_LC601_CMD : fbDPT_Switch_pro;
    M1_168_5F201_RT601_SP : fbDPT_Value_Temp_pro;
    M1_169_5F201_RT601_SP_FB : fbDPT_Value_Temp_pro;
    M1_170_5F202_RB601_V : fbDPT_Switch_pro;  (* 5F202 *)
    M1_171_5F202_RB602_V : fbDPT_Switch_pro;
    M1_172_5F202_RB603_V : fbDPT_Switch_pro;
    M1_173_5F202_RB604_V : fbDPT_Switch_pro;
    M1_174_5F202_RB605_V : fbDPT_Switch_pro;
    M1_175_5F202_RB601_HVAC : fbDPT_Switch_pro;
    M1_176_5F202_RB602_HVAC : fbDPT_Switch_pro;
    M1_177_5F202_RB603_HVAC : fbDPT_Switch_pro;
    M1_178_5F202_RB604_HVAC : fbDPT_Switch_pro;
    M1_179_5F202_RB605_HVAC : fbDPT_Switch_pro;
    M1_180_5F202_RT601_CT : fbDPT_Value_Temp_pro;
    M1_181_5F202_RT602_CT : fbDPT_Value_Temp_pro;
    M1_182_5F202_RY601_CV : fbDPT_Value_AirQuality_pro;
    M1_183_5F202_LH601_OP : fbDPT_Scaling_pro;
    M1_184_5F202_LH601_CMD : fbDPT_Switch_pro;
    M1_185_5F202_LC601_OP : fbDPT_Scaling_pro;
    M1_186_5F202_LC601_CMD : fbDPT_Switch_pro;
    M1_187_5F202_RT601_SP : fbDPT_Value_Temp_pro;
    M1_188_5F202_RT601_SP_FB : fbDPT_Value_Temp_pro;
    M1_189_5F301_RB601_V : fbDPT_Switch_pro;  (* 5F301 *)
    M1_190_5F301_RB601_HVAC : fbDPT_Switch_pro;
    M1_191_5F301_RT601_CT : fbDPT_Value_Temp_pro;
    M1_192_5F301_RY601_CV : fbDPT_Value_AirQuality_pro;
    M1_193_5F301_LH601_OP : fbDPT_Scaling_pro;
    M1_194_5F301_LH601_CMD : fbDPT_Switch_pro;
    M1_195_5F301_LC601_OP : fbDPT_Scaling_pro;
    M1_196_5F301_LC601_CMD : fbDPT_Switch_pro;
    M1_197_5F301_RT601_SP : fbDPT_Value_Temp_pro;
    M1_198_5F301_RT601_SP_FB : fbDPT_Value_Temp_pro;
    M1_199_5F302_RB601_V : fbDPT_Switch_pro;  (* 5F302 *)
    M1_200_5F302_RB601_HVAC : fbDPT_Switch_pro;
    M1_201_5F302_RT601_CT : fbDPT_Value_Temp_pro;
    M1_202_5F302_RY601_CV : fbDPT_Value_AirQuality_pro;
    M1_203_5F302_LH601_OP : fbDPT_Scaling_pro;
    M1_204_5F302_LH601_CMD : fbDPT_Switch_pro;
    M1_205_5F302_LC601_OP : fbDPT_Scaling_pro;
    M1_206_5F302_LC601_CMD : fbDPT_Switch_pro;
    M1_207_5F302_RT601_SP : fbDPT_Value_Temp_pro;
    M1_208_5F302_RT601_SP_FB : fbDPT_Value_Temp_pro;
    M1_209_5G201_RB601_V : fbDPT_Switch_pro;  (* 5G201 *)
    M1_210_5G201_RB601_HVAC : fbDPT_Switch_pro;
    M1_211_5G201_RT601_CT : fbDPT_Value_Temp_pro;
    M1_212_5G201_RY601_CV : fbDPT_Value_AirQuality_pro;
    M1_213_5G201_LH601_OP : fbDPT_Scaling_pro;
    M1_214_5G201_LH601_CMD : fbDPT_Switch_pro;
    M1_215_5G201_LC601_OP : fbDPT_Scaling_pro;
    M1_216_5G201_LC601_CMD : fbDPT_Switch_pro;
    M1_217_5G201_RT601_SP : fbDPT_Value_Temp_pro;
    M1_218_5G201_RT601_SP_FB : fbDPT_Value_Temp_pro;
    M1_219_5G202_RB601_V : fbDPT_Switch_pro;  (* 5G202 *)
    M1_220_5G202_RB601_HVAC : fbDPT_Switch_pro;
    M1_221_5G202_RT601_CT : fbDPT_Value_Temp_pro;
    M1_222_5G202_RY601_CV : fbDPT_Value_AirQuality_pro;
    M1_223_5G202_LH601_OP : fbDPT_Scaling_pro;
    M1_224_5G202_LH601_CMD : fbDPT_Switch_pro;
    M1_225_5G202_LC601_OP : fbDPT_Scaling_pro;
    M1_226_5G202_LC601_CMD : fbDPT_Switch_pro;
    M1_227_5G202_RT601_SP : fbDPT_Value_Temp_pro;
    M1_228_5G202_RT601_SP_FB : fbDPT_Value_Temp_pro;
    M1_229_5H301_RB601_V : fbDPT_Switch_pro;  (* 5H301 *)
    M1_230_5H301_RB601_HVAC : fbDPT_Switch_pro;
    M1_231_5H301_RT601_CT : fbDPT_Value_Temp_pro;
    M1_232_5H301_RY601_CV : fbDPT_Value_AirQuality_pro;
    M1_233_5H301_LH601_OP : fbDPT_Scaling_pro;
    M1_234_5H301_LH601_CMD : fbDPT_Switch_pro;
    M1_235_5H301_LC601_OP : fbDPT_Scaling_pro;
    M1_236_5H301_LC601_CMD : fbDPT_Switch_pro;
    M1_237_5H301_RT601_SP : fbDPT_Value_Temp_pro;
    M1_238_5H301_RT601_SP_FB : fbDPT_Value_Temp_pro;
    M1_239_5H302_RB601_V : fbDPT_Switch_pro;  (* 5H302 *)
    M1_240_5H302_RB601_HVAC : fbDPT_Switch_pro;
    M1_241_5H302_RT601_CT : fbDPT_Value_Temp_pro;
    M1_242_5H302_RY601_CV : fbDPT_Value_AirQuality_pro;
    M1_243_5H302_LH601_OP : fbDPT_Scaling_pro;
    M1_244_5H302_LH601_CMD : fbDPT_Switch_pro;
    M1_245_5H302_LC601_OP : fbDPT_Scaling_pro;
    M1_246_5H302_LC601_CMD : fbDPT_Switch_pro;
    M1_247_5H302_RT601_SP : fbDPT_Value_Temp_pro;
    M1_248_5H302_RT601_SP_FB : fbDPT_Value_Temp_pro;
  END_VAR

(* CFC diagram, written out as Structured Text *)
(* KNX Master *)
KNX_master_1(I_Port := IoConfig_Globals.KNX_EIB_TP1_Interface, bPortKNX := 1);
STLV80_563.STLV80_A_563_KNX_Card_1_Status := KNX_master_1.sStatus = 'OK';
(* Rom 5A201 *)
(* RB601_V *)
M1_001_5A201_RB601_V(bPortKNX := 1, dwIndex_DPT := 1, typDPT := typDPT);
STLV80_563.STLV80_A_563_5A201.RB601_V := M1_001_5A201_RB601_V.xSwitch_OUT;
(* Rom 5A202 *)
(* RB601_V *)
(* RB601_HVAC *)
M1_002_5A202_RB601_V(bPortKNX := 1, dwIndex_DPT := 2, typDPT := typDPT);
STLV80_563.STLV80_A_563_5A202.RB601_V := M1_002_5A202_RB601_V.xSwitch_OUT;
M1_003_5A202_RB601_HVAC(bPortKNX := 1, dwIndex_DPT := 3, typDPT := typDPT);
STLV80_563.STLV80_A_563_5A202.RB601_HVAC := M1_003_5A202_RB601_HVAC.xSwitch_OUT;
(* Rom 5A301 *)
(* RB601_V *)
(* RB601_HVAC *)
M1_004_5A301_RB601_V(bPortKNX := 1, dwIndex_DPT := 4, typDPT := typDPT);
STLV80_563.STLV80_A_563_5A301.RB601_V := M1_004_5A301_RB601_V.xSwitch_OUT;
M1_005_5A301_RB601_HVAC(bPortKNX := 1, dwIndex_DPT := 5, typDPT := typDPT);
STLV80_563.STLV80_A_563_5A301.RB601_HVAC := M1_005_5A301_RB601_HVAC.xSwitch_OUT;
(* RT601_CT *)
M1_006_5A301_RT601_CT(bPortKNX := 1, dwIndex_DPT := 6, typDPT := typDPT);
STLV80_563.STLV80_A_563_5A301.RT601_CT := M1_006_5A301_RT601_CT.rValue_OUT;
(* Rom 5A302 *)
(* RB601_V *)
(* RB601_HVAC *)
M1_007_5A302_RB601_V(bPortKNX := 1, dwIndex_DPT := 7, typDPT := typDPT);
STLV80_563.STLV80_A_563_5A302.RB601_V := M1_007_5A302_RB601_V.xSwitch_OUT;
M1_008_5A302_RB601_HVAC(bPortKNX := 1, dwIndex_DPT := 8, typDPT := typDPT);
STLV80_563.STLV80_A_563_5A302.RB601_HVAC := M1_008_5A302_RB601_HVAC.xSwitch_OUT;
(* RT601_CT *)
(* RY601_CV *)
M1_009_5A302_RT601_CT(bPortKNX := 1, dwIndex_DPT := 9, typDPT := typDPT);
STLV80_563.STLV80_A_563_5A302.RT601_CT := M1_009_5A302_RT601_CT.rValue_OUT;
M1_010_5A302_RY601_CV(bPortKNX := 1, dwIndex_DPT := 10, typDPT := typDPT);
STLV80_563.STLV80_A_563_5A302.RY601_CV := M1_010_5A302_RY601_CV.rValue_OUT;
(* Rom 5B201 *)
(* RB601_V *)
(* RB601_HVAC *)
M1_011_5B201_RB601_V(bPortKNX := 1, dwIndex_DPT := 11, typDPT := typDPT);
STLV80_563.STLV80_A_563_5B201.RB601_V := M1_011_5B201_RB601_V.xSwitch_OUT;
M1_012_5B201_RB601_HVAC(bPortKNX := 1, dwIndex_DPT := 12, typDPT := typDPT);
STLV80_563.STLV80_A_563_5B201.RB601_HVAC := M1_012_5B201_RB601_HVAC.xSwitch_OUT;
(* RT601_CT *)
(* LH601_OP *)
M1_013_5B201_RT601_CT(bPortKNX := 1, dwIndex_DPT := 13, typDPT := typDPT);
STLV80_563.STLV80_A_563_5B201.RT601_CT := M1_013_5B201_RT601_CT.rValue_OUT;
M1_014_5B201_LH601_OP(bPortKNX := 1, dwIndex_DPT := 14, rValue_IN := STLV80_563.STLV80_A_563_5B201.LH601_OP, xUpdate_KNX := i = 0, typDPT := typDPT);
(* Rom 5B202 *)
(* RB601_V *)
(* RB601_HVAC *)
M1_015_5B202_RB601_V(bPortKNX := 1, dwIndex_DPT := 15, typDPT := typDPT);
STLV80_563.STLV80_A_563_5B202.RB601_V := M1_015_5B202_RB601_V.xSwitch_OUT;
M1_016_5B202_RB601_HVAC(bPortKNX := 1, dwIndex_DPT := 16, typDPT := typDPT);
STLV80_563.STLV80_A_563_5B202.RB601_HVAC := M1_016_5B202_RB601_HVAC.xSwitch_OUT;
(* RT601_CT *)
(* LH601_OP *)
M1_017_5B202_RT601_CT(bPortKNX := 1, dwIndex_DPT := 17, typDPT := typDPT);
STLV80_563.STLV80_A_563_5B202.RT601_CT := M1_017_5B202_RT601_CT.rValue_OUT;
M1_018_5B202_LH601_OP(bPortKNX := 1, dwIndex_DPT := 18, rValue_IN := STLV80_563.STLV80_A_563_5B202.LH601_OP, xUpdate_KNX := i = 1, typDPT := typDPT);
(* LH601_CMD *)
M1_019_5B202_LH601_CMD(bPortKNX := 1, dwIndex_DPT := 19, xSwitch_IN := STLV80_563.STLV80_A_563_5B202.LH601_CMD, xUpdate_KNX := i = 2, typDPT := typDPT);
(* Rom 5B301 *)
(* RB601_V *)
(* RB601_HVAC *)
M1_020_5B301_RB601_V(bPortKNX := 1, dwIndex_DPT := 20, typDPT := typDPT);
STLV80_563.STLV80_A_563_5B301.RB601_V := M1_020_5B301_RB601_V.xSwitch_OUT;
M1_021_5B301_RB601_HVAC(bPortKNX := 1, dwIndex_DPT := 21, typDPT := typDPT);
STLV80_563.STLV80_A_563_5B301.RB601_HVAC := M1_021_5B301_RB601_HVAC.xSwitch_OUT;
(* RT601_CT *)
(* LH601_OP *)
M1_022_5B301_RT601_CT(bPortKNX := 1, dwIndex_DPT := 22, typDPT := typDPT);
STLV80_563.STLV80_A_563_5B301.RT601_CT := M1_022_5B301_RT601_CT.rValue_OUT;
M1_023_5B301_LH601_OP(bPortKNX := 1, dwIndex_DPT := 23, rValue_IN := STLV80_563.STLV80_A_563_5B301.LH601_OP, xUpdate_KNX := i = 3, typDPT := typDPT);
(* LH601_CMD *)
(* LC601_OP *)
M1_024_5B301_LH601_CMD(bPortKNX := 1, dwIndex_DPT := 24, xSwitch_IN := STLV80_563.STLV80_A_563_5B301.LH601_CMD, xUpdate_KNX := i = 4, typDPT := typDPT);
M1_025_5B301_LC601_OP(bPortKNX := 1, dwIndex_DPT := 25, rValue_IN := STLV80_563.STLV80_A_563_5B301.LC601_OP, xUpdate_KNX := i = 5, typDPT := typDPT);
(* Rom 5B302 *)
(* RB601_V *)
(* RB601_HVAC *)
M1_026_5B302_RB601_V(bPortKNX := 1, dwIndex_DPT := 26, typDPT := typDPT);
STLV80_563.STLV80_A_563_5B302.RB601_V := M1_026_5B302_RB601_V.xSwitch_OUT;
M1_027_5B302_RB601_HVAC(bPortKNX := 1, dwIndex_DPT := 27, typDPT := typDPT);
STLV80_563.STLV80_A_563_5B302.RB601_HVAC := M1_027_5B302_RB601_HVAC.xSwitch_OUT;
(* RT601_CT *)
(* RY601_CV *)
M1_028_5B302_RT601_CT(bPortKNX := 1, dwIndex_DPT := 28, typDPT := typDPT);
STLV80_563.STLV80_A_563_5B302.RT601_CT := M1_028_5B302_RT601_CT.rValue_OUT;
M1_029_5B302_RY601_CV(bPortKNX := 1, dwIndex_DPT := 29, typDPT := typDPT);
STLV80_563.STLV80_A_563_5B302.RY601_CV := M1_029_5B302_RY601_CV.rValue_OUT;
(* LH601_OP *)
(* LH601_CMD *)
M1_030_5B302_LH601_OP(bPortKNX := 1, dwIndex_DPT := 30, rValue_IN := STLV80_563.STLV80_A_563_5B302.LH601_OP, xUpdate_KNX := i = 6, typDPT := typDPT);
M1_031_5B302_LH601_CMD(bPortKNX := 1, dwIndex_DPT := 31, xSwitch_IN := STLV80_563.STLV80_A_563_5B302.LH601_CMD, xUpdate_KNX := i = 7, typDPT := typDPT);
(* LC601_OP *)
(* LC601_CMD *)
M1_032_5B302_LC601_OP(bPortKNX := 1, dwIndex_DPT := 32, rValue_IN := STLV80_563.STLV80_A_563_5B302.LC601_OP, xUpdate_KNX := i = 8, typDPT := typDPT);
M1_033_5B302_LC601_CMD(bPortKNX := 1, dwIndex_DPT := 33, xSwitch_IN := STLV80_563.STLV80_A_563_5B302.LC601_CMD, xUpdate_KNX := i = 9, typDPT := typDPT);
(* Rom 5C201 *)
(* RB601_V *)
(* RB601_HVAC *)
M1_034_5C201_RB601_V(bPortKNX := 1, dwIndex_DPT := 34, typDPT := typDPT);
STLV80_563.STLV80_A_563_5C201.RB601_V := M1_034_5C201_RB601_V.xSwitch_OUT;
M1_035_5C201_RB601_HVAC(bPortKNX := 1, dwIndex_DPT := 35, typDPT := typDPT);
STLV80_563.STLV80_A_563_5C201.RB601_HVAC := M1_035_5C201_RB601_HVAC.xSwitch_OUT;
(* RT601_CT *)
(* LH601_OP *)
M1_036_5C201_RT601_CT(bPortKNX := 1, dwIndex_DPT := 36, typDPT := typDPT);
STLV80_563.STLV80_A_563_5C201.RT601_CT := M1_036_5C201_RT601_CT.rValue_OUT;
M1_037_5C201_LH601_OP(bPortKNX := 1, dwIndex_DPT := 37, rValue_IN := STLV80_563.STLV80_A_563_5C201.LH601_OP, xUpdate_KNX := i = 10, typDPT := typDPT);
(* LC601_OP *)
(* LC601_CMD *)
M1_038_5C201_LC601_OP(bPortKNX := 1, dwIndex_DPT := 38, rValue_IN := STLV80_563.STLV80_A_563_5C201.LC601_OP, xUpdate_KNX := i = 11, typDPT := typDPT);
M1_039_5C201_LC601_CMD(bPortKNX := 1, dwIndex_DPT := 39, xSwitch_IN := STLV80_563.STLV80_A_563_5C201.LC601_CMD, xUpdate_KNX := i = 12, typDPT := typDPT);
(* RT601_SP *)
M1_040_5C201_RT601_SP(bPortKNX := 1, dwIndex_DPT := 40, rValue_IN := STLV80_563.STLV80_A_563_5C201.RT601_SP_D, xUpdate_KNX := NOT STLV80_563.STLV80_A_563_5C201.RB601_HVAC, typDPT := typDPT);
(* Rom 5C202 *)
(* RB601_V *)
(* RB601_HVAC *)
M1_041_5C202_RB601_V(bPortKNX := 1, dwIndex_DPT := 41, typDPT := typDPT);
STLV80_563.STLV80_A_563_5C202.RB601_V := M1_041_5C202_RB601_V.xSwitch_OUT;
M1_042_5C202_RB601_HVAC(bPortKNX := 1, dwIndex_DPT := 42, typDPT := typDPT);
STLV80_563.STLV80_A_563_5C202.RB601_HVAC := M1_042_5C202_RB601_HVAC.xSwitch_OUT;
(* RT601_CT *)
(* RY601_CV *)
M1_043_5C202_RT601_CT(bPortKNX := 1, dwIndex_DPT := 43, typDPT := typDPT);
STLV80_563.STLV80_A_563_5C202.RT601_CT := M1_043_5C202_RT601_CT.rValue_OUT;
M1_044_5C202_RY601_CV(bPortKNX := 1, dwIndex_DPT := 44, typDPT := typDPT);
STLV80_563.STLV80_A_563_5C202.RY601_CV := M1_044_5C202_RY601_CV.rValue_OUT;
(* LH601_OP *)
(* LC601_OP *)
M1_045_5C202_LH601_OP(bPortKNX := 1, dwIndex_DPT := 45, rValue_IN := STLV80_563.STLV80_A_563_5C202.LH601_OP, xUpdate_KNX := i = 13, typDPT := typDPT);
M1_046_5C202_LC601_OP(bPortKNX := 1, dwIndex_DPT := 46, rValue_IN := STLV80_563.STLV80_A_563_5C202.LC601_OP, xUpdate_KNX := i = 14, typDPT := typDPT);
(* RT601_SP *)
(* RT601_SP Feedback *)
M1_047_5C202_RT601_SP(bPortKNX := 1, dwIndex_DPT := 47, rValue_IN := STLV80_563.STLV80_A_563_5C202.RT601_SP_D, xUpdate_KNX := NOT STLV80_563.STLV80_A_563_5C202.RB601_HVAC, typDPT := typDPT);
M1_048_5C202_RT601_SP_FB(bPortKNX := 1, dwIndex_DPT := 48, typDPT := typDPT);
STLV80_563.STLV80_A_563_5C202.RT601_SP_IN := M1_048_5C202_RT601_SP_FB.rValue_OUT;
(* Rom 5C301 *)
(* RB601_V *)
(* RB601_HVAC *)
M1_049_5C301_RB601_V(bPortKNX := 1, dwIndex_DPT := 49, typDPT := typDPT);
STLV80_563.STLV80_A_563_5C301.RB601_V := M1_049_5C301_RB601_V.xSwitch_OUT;
M1_050_5C301_RB601_HVAC(bPortKNX := 1, dwIndex_DPT := 50, typDPT := typDPT);
STLV80_563.STLV80_A_563_5C301.RB601_HVAC := M1_050_5C301_RB601_HVAC.xSwitch_OUT;
(* RT601_CT *)
(* RY601_CV *)
M1_051_5C301_RT601_CT(bPortKNX := 1, dwIndex_DPT := 51, typDPT := typDPT);
STLV80_563.STLV80_A_563_5C301.RT601_CT := M1_051_5C301_RT601_CT.rValue_OUT;
M1_052_5C301_RY601_CV(bPortKNX := 1, dwIndex_DPT := 52, typDPT := typDPT);
STLV80_563.STLV80_A_563_5C301.RY601_CV := M1_052_5C301_RY601_CV.rValue_OUT;
(* LH601_OP *)
(* LH601_CMD *)
M1_053_5C301_LH601_OP(bPortKNX := 1, dwIndex_DPT := 53, rValue_IN := STLV80_563.STLV80_A_563_5C301.LH601_OP, xUpdate_KNX := i = 15, typDPT := typDPT);
M1_054_5C301_LH601_CMD(bPortKNX := 1, dwIndex_DPT := 54, xSwitch_IN := STLV80_563.STLV80_A_563_5C301.LH601_CMD, xUpdate_KNX := i = 16, typDPT := typDPT);
(* LC601_OP *)
(* LC601_CMD *)
M1_055_5C301_LC601_OP(bPortKNX := 1, dwIndex_DPT := 55, rValue_IN := STLV80_563.STLV80_A_563_5C301.LC601_OP, xUpdate_KNX := i = 17, typDPT := typDPT);
M1_056_5C301_LC601_CMD(bPortKNX := 1, dwIndex_DPT := 56, xSwitch_IN := STLV80_563.STLV80_A_563_5C301.LC601_CMD, xUpdate_KNX := i = 18, typDPT := typDPT);
(* Rom 5C302 *)
(* RB601_V *)
(* RB602_V *)
M1_057_5C302_RB601_V(bPortKNX := 1, dwIndex_DPT := 57, typDPT := typDPT);
STLV80_563.STLV80_A_563_5C302.RB601_V := M1_057_5C302_RB601_V.xSwitch_OUT;
M1_058_5C302_RB602_V(bPortKNX := 1, dwIndex_DPT := 58, typDPT := typDPT);
STLV80_563.STLV80_A_563_5C302.RB602_V := M1_058_5C302_RB602_V.xSwitch_OUT;
(* RB601_HVAC *)
(* RT601_CT *)
M1_059_5C302_RB601_HVAC(bPortKNX := 1, dwIndex_DPT := 59, typDPT := typDPT);
STLV80_563.STLV80_A_563_5C302.RB601_HVAC := M1_059_5C302_RB601_HVAC.xSwitch_OUT;
M1_060_5C302_RT601_CT(bPortKNX := 1, dwIndex_DPT := 60, typDPT := typDPT);
STLV80_563.STLV80_A_563_5C302.RT601_CT := M1_060_5C302_RT601_CT.rValue_OUT;
(* RY601_CV *)
(* LH601_OP *)
M1_061_5C302_RY601_CV(bPortKNX := 1, dwIndex_DPT := 61, typDPT := typDPT);
STLV80_563.STLV80_A_563_5C302.RY601_CV := M1_061_5C302_RY601_CV.rValue_OUT;
M1_062_5C302_LH601_OP(bPortKNX := 1, dwIndex_DPT := 62, rValue_IN := STLV80_563.STLV80_A_563_5C302.LH601_OP, xUpdate_KNX := i = 19, typDPT := typDPT);
(* LH601_CMD *)
(* LC601_OP *)
M1_063_5C302_LH601_CMD(bPortKNX := 1, dwIndex_DPT := 63, xSwitch_IN := STLV80_563.STLV80_A_563_5C302.LH601_CMD, xUpdate_KNX := i = 20, typDPT := typDPT);
M1_064_5C302_LC601_OP(bPortKNX := 1, dwIndex_DPT := 64, rValue_IN := STLV80_563.STLV80_A_563_5C302.LC601_OP, xUpdate_KNX := i = 21, typDPT := typDPT);
(* LC601_CMD *)
(* RT601_SP *)
M1_065_5C302_LC601_CMD(bPortKNX := 1, dwIndex_DPT := 65, xSwitch_IN := STLV80_563.STLV80_A_563_5C302.LC601_CMD, xUpdate_KNX := i = 22, typDPT := typDPT);
M1_066_5C302_RT601_SP(bPortKNX := 1, dwIndex_DPT := 66, rValue_IN := STLV80_563.STLV80_A_563_5C302.RT601_SP_D, xUpdate_KNX := NOT STLV80_563.STLV80_A_563_5C302.RB601_HVAC, typDPT := typDPT);
(* RT601_SP Feedback *)
M1_067_5C302_RT601_SP_FB(bPortKNX := 1, dwIndex_DPT := 67, typDPT := typDPT);
STLV80_563.STLV80_A_563_5C302.RT601_SP_IN := M1_067_5C302_RT601_SP_FB.rValue_OUT;
(* Rom 5D201 *)
(* RB601_V *)
(* RB601_HVAC *)
M1_068_5D201_RB601_V(bPortKNX := 1, dwIndex_DPT := 68, typDPT := typDPT);
STLV80_563.STLV80_A_563_5D201.RB601_V := M1_068_5D201_RB601_V.xSwitch_OUT;
M1_069_5D201_RB601_HVAC(bPortKNX := 1, dwIndex_DPT := 69, typDPT := typDPT);
STLV80_563.STLV80_A_563_5D201.RB601_HVAC := M1_069_5D201_RB601_HVAC.xSwitch_OUT;
(* RB602_HVAC *)
(* RT601_CT *)
M1_070_5D201_RB602_HVAC(bPortKNX := 1, dwIndex_DPT := 70, typDPT := typDPT);
STLV80_563.STLV80_A_563_5D201.RB602_HVAC := M1_070_5D201_RB602_HVAC.xSwitch_OUT;
M1_071_5D201_RT601_CT(bPortKNX := 1, dwIndex_DPT := 71, typDPT := typDPT);
STLV80_563.STLV80_A_563_5D201.RT601_CT := M1_071_5D201_RT601_CT.rValue_OUT;
(* RY601_CV *)
(* LH601_OP *)
M1_072_5D201_RY601_CV(bPortKNX := 1, dwIndex_DPT := 72, typDPT := typDPT);
STLV80_563.STLV80_A_563_5D201.RY601_CV := M1_072_5D201_RY601_CV.rValue_OUT;
M1_073_5D201_LH601_OP(bPortKNX := 1, dwIndex_DPT := 73, rValue_IN := STLV80_563.STLV80_A_563_5D201.LH601_OP, xUpdate_KNX := i = 23, typDPT := typDPT);
(* LH601_CMD *)
(* LC601_OP *)
M1_074_5D201_LH601_CMD(bPortKNX := 1, dwIndex_DPT := 74, xSwitch_IN := STLV80_563.STLV80_A_563_5D201.LH601_CMD, xUpdate_KNX := i = 24, typDPT := typDPT);
M1_075_5D201_LC601_OP(bPortKNX := 1, dwIndex_DPT := 75, rValue_IN := STLV80_563.STLV80_A_563_5D201.LC601_OP, xUpdate_KNX := i = 25, typDPT := typDPT);
(* LC601_CMD *)
(* RT601_SP *)
M1_076_5D201_LC601_CMD(bPortKNX := 1, dwIndex_DPT := 76, xSwitch_IN := STLV80_563.STLV80_A_563_5D201.LC601_CMD, xUpdate_KNX := i = 26, typDPT := typDPT);
M1_077_5D201_RT601_SP(bPortKNX := 1, dwIndex_DPT := 77, rValue_IN := STLV80_563.STLV80_A_563_5D201.RT601_SP_D, xUpdate_KNX := NOT STLV80_563.STLV80_A_563_5D201.RB601_HVAC, typDPT := typDPT);
(* RT601_SP Feedback *)
M1_078_5D201_RT601_SP_FB(bPortKNX := 1, dwIndex_DPT := 78, typDPT := typDPT);
STLV80_563.STLV80_A_563_5D201.RT601_SP_IN := M1_078_5D201_RT601_SP_FB.rValue_OUT;
(* Rom 5D202 *)
(* RB601_V *)
(* RB601_HVAC *)
M1_079_5D202_RB601_V(bPortKNX := 1, dwIndex_DPT := 79, typDPT := typDPT);
STLV80_563.STLV80_A_563_5D202.RB601_V := M1_079_5D202_RB601_V.xSwitch_OUT;
M1_080_5D202_RB601_HVAC(bPortKNX := 1, dwIndex_DPT := 80, typDPT := typDPT);
STLV80_563.STLV80_A_563_5D202.RB601_HVAC := M1_080_5D202_RB601_HVAC.xSwitch_OUT;
(* RT601_CT *)
(* RT602_CT *)
M1_081_5D202_RT601_CT(bPortKNX := 1, dwIndex_DPT := 81, typDPT := typDPT);
STLV80_563.STLV80_A_563_5D202.RT601_CT := M1_081_5D202_RT601_CT.rValue_OUT;
M1_082_5D202_RT602_CT(bPortKNX := 1, dwIndex_DPT := 82, typDPT := typDPT);
STLV80_563.STLV80_A_563_5D202.RT602_CT := M1_082_5D202_RT602_CT.rValue_OUT;
(* RY601_CV *)
(* LH601_OP *)
M1_083_5D202_RY601_CV(bPortKNX := 1, dwIndex_DPT := 83, typDPT := typDPT);
STLV80_563.STLV80_A_563_5D202.RY601_CV := M1_083_5D202_RY601_CV.rValue_OUT;
M1_084_5D202_LH601_OP(bPortKNX := 1, dwIndex_DPT := 84, rValue_IN := STLV80_563.STLV80_A_563_5D202.LH601_OP, xUpdate_KNX := i = 27, typDPT := typDPT);
(* LH601_CMD *)
(* LC601_OP *)
M1_085_5D202_LH601_CMD(bPortKNX := 1, dwIndex_DPT := 85, xSwitch_IN := STLV80_563.STLV80_A_563_5D202.LH601_CMD, xUpdate_KNX := i = 28, typDPT := typDPT);
M1_086_5D202_LC601_OP(bPortKNX := 1, dwIndex_DPT := 86, rValue_IN := STLV80_563.STLV80_A_563_5D202.LC601_OP, xUpdate_KNX := i = 29, typDPT := typDPT);
(* LC601_CMD *)
(* RT601_SP *)
M1_087_5D202_LC601_CMD(bPortKNX := 1, dwIndex_DPT := 87, xSwitch_IN := STLV80_563.STLV80_A_563_5D202.LC601_CMD, xUpdate_KNX := i = 30, typDPT := typDPT);
M1_088_5D202_RT601_SP(bPortKNX := 1, dwIndex_DPT := 88, rValue_IN := STLV80_563.STLV80_A_563_5D202.RT601_SP_D, xUpdate_KNX := NOT STLV80_563.STLV80_A_563_5D202.RB601_HVAC, typDPT := typDPT);
(* RT601_SP Feedback *)
M1_089_5D202_RT601_SP_FB(bPortKNX := 1, dwIndex_DPT := 89, typDPT := typDPT);
STLV80_563.STLV80_A_563_5D202.RT601_SP_IN := M1_089_5D202_RT601_SP_FB.rValue_OUT;
(* Rom 5D301 *)
(* RB601_V *)
(* RB601_HVAC *)
M1_090_5D301_RB601_V(bPortKNX := 1, dwIndex_DPT := 90, typDPT := typDPT);
STLV80_563.STLV80_A_563_5D301.RB601_V := M1_090_5D301_RB601_V.xSwitch_OUT;
M1_091_5D301_RB601_HVAC(bPortKNX := 1, dwIndex_DPT := 91, typDPT := typDPT);
STLV80_563.STLV80_A_563_5D301.RB601_HVAC := M1_091_5D301_RB601_HVAC.xSwitch_OUT;
(* RT601_CT *)
(* RY601_CV *)
M1_092_5D301_RT601_CT(bPortKNX := 1, dwIndex_DPT := 92, typDPT := typDPT);
STLV80_563.STLV80_A_563_5D301.RT601_CT := M1_092_5D301_RT601_CT.rValue_OUT;
M1_093_5D301_RY601_CV(bPortKNX := 1, dwIndex_DPT := 93, typDPT := typDPT);
STLV80_563.STLV80_A_563_5D301.RY601_CV := M1_093_5D301_RY601_CV.rValue_OUT;
(* RY602_CV *)
(* LH601_OP *)
M1_094_5D301_RY602_CV(bPortKNX := 1, dwIndex_DPT := 94, typDPT := typDPT);
STLV80_563.STLV80_A_563_5D301.RY602_CV := M1_094_5D301_RY602_CV.rValue_OUT;
M1_095_5D301_LH601_OP(bPortKNX := 1, dwIndex_DPT := 95, rValue_IN := STLV80_563.STLV80_A_563_5D301.LH601_OP, xUpdate_KNX := i = 31, typDPT := typDPT);
(* LH601_CMD *)
(* LC601_OP *)
M1_096_5D301_LH601_CMD(bPortKNX := 1, dwIndex_DPT := 96, xSwitch_IN := STLV80_563.STLV80_A_563_5D301.LH601_CMD, xUpdate_KNX := i = 32, typDPT := typDPT);
M1_097_5D301_LC601_OP(bPortKNX := 1, dwIndex_DPT := 97, rValue_IN := STLV80_563.STLV80_A_563_5D301.LC601_OP, xUpdate_KNX := i = 33, typDPT := typDPT);
(* LC601_CMD *)
(* RT601_SP *)
M1_098_5D301_LC601_CMD(bPortKNX := 1, dwIndex_DPT := 98, xSwitch_IN := STLV80_563.STLV80_A_563_5D301.LC601_CMD, xUpdate_KNX := i = 34, typDPT := typDPT);
M1_099_5D301_RT601_SP(bPortKNX := 1, dwIndex_DPT := 99, rValue_IN := STLV80_563.STLV80_A_563_5D301.RT601_SP_D, xUpdate_KNX := NOT STLV80_563.STLV80_A_563_5D301.RB601_HVAC, typDPT := typDPT);
(* RT601_SP Feedback *)
M1_100_5D301_RT601_SP_FB(bPortKNX := 1, dwIndex_DPT := 100, typDPT := typDPT);
STLV80_563.STLV80_A_563_5D301.RT601_SP_IN := M1_100_5D301_RT601_SP_FB.rValue_OUT;
(* Rom 5D302 *)
(* RB601_V *)
(* RB601_HVAC *)
M1_101_5D302_RB601_V(bPortKNX := 1, dwIndex_DPT := 101, typDPT := typDPT);
STLV80_563.STLV80_A_563_5D302.RB601_V := M1_101_5D302_RB601_V.xSwitch_OUT;
M1_102_5D302_RB601_HVAC(bPortKNX := 1, dwIndex_DPT := 102, typDPT := typDPT);
STLV80_563.STLV80_A_563_5D302.RB601_HVAC := M1_102_5D302_RB601_HVAC.xSwitch_OUT;
(* RT601_CT *)
(* RY601_CV *)
M1_103_5D302_RT601_CT(bPortKNX := 1, dwIndex_DPT := 103, typDPT := typDPT);
STLV80_563.STLV80_A_563_5D302.RT601_CT := M1_103_5D302_RT601_CT.rValue_OUT;
M1_104_5D302_RY601_CV(bPortKNX := 1, dwIndex_DPT := 104, typDPT := typDPT);
STLV80_563.STLV80_A_563_5D302.RY601_CV := M1_104_5D302_RY601_CV.rValue_OUT;
(* LH601_OP *)
(* LH602_OP *)
M1_105_5D302_LH601_OP(bPortKNX := 1, dwIndex_DPT := 105, rValue_IN := STLV80_563.STLV80_A_563_5D302.LH601_OP, xUpdate_KNX := i = 35, typDPT := typDPT);
M1_106_5D302_LH602_OP(bPortKNX := 1, dwIndex_DPT := 106, rValue_IN := STLV80_563.STLV80_A_563_5D302.LH602_OP, xUpdate_KNX := i = 36, typDPT := typDPT);
(* LH601_CMD *)
(* LC601_OP *)
M1_107_5D302_LH601_CMD(bPortKNX := 1, dwIndex_DPT := 107, xSwitch_IN := STLV80_563.STLV80_A_563_5D302.LH601_CMD, xUpdate_KNX := i = 37, typDPT := typDPT);
M1_108_5D302_LC601_OP(bPortKNX := 1, dwIndex_DPT := 108, rValue_IN := STLV80_563.STLV80_A_563_5D302.LC601_OP, xUpdate_KNX := i = 38, typDPT := typDPT);
(* LC601_CMD *)
(* RT601_SP *)
M1_109_5D302_LC601_CMD(bPortKNX := 1, dwIndex_DPT := 109, xSwitch_IN := STLV80_563.STLV80_A_563_5D302.LC601_CMD, xUpdate_KNX := i = 39, typDPT := typDPT);
M1_110_5D302_RT601_SP(bPortKNX := 1, dwIndex_DPT := 110, rValue_IN := STLV80_563.STLV80_A_563_5D302.RT601_SP_D, xUpdate_KNX := NOT STLV80_563.STLV80_A_563_5D302.RB601_HVAC, typDPT := typDPT);
(* RT601_SP Feedback *)
M1_111_5D302_RT601_SP_FB(bPortKNX := 1, dwIndex_DPT := 111, typDPT := typDPT);
STLV80_563.STLV80_A_563_5D302.RT601_SP_IN := M1_111_5D302_RT601_SP_FB.rValue_OUT;
(* Rom 5E201 *)
(* RB601_V *)
(* RB601_HVAC *)
M1_112_5E201_RB601_V(bPortKNX := 1, dwIndex_DPT := 112, typDPT := typDPT);
STLV80_563.STLV80_A_563_5E201.RB601_V := M1_112_5E201_RB601_V.xSwitch_OUT;
M1_113_5E201_RB601_HVAC(bPortKNX := 1, dwIndex_DPT := 113, typDPT := typDPT);
STLV80_563.STLV80_A_563_5E201.RB601_HVAC := M1_113_5E201_RB601_HVAC.xSwitch_OUT;
(* RT601_CT *)
(* RY601_CV *)
M1_114_5E201_RT601_CT(bPortKNX := 1, dwIndex_DPT := 114, typDPT := typDPT);
STLV80_563.STLV80_A_563_5E201.RT601_CT := M1_114_5E201_RT601_CT.rValue_OUT;
M1_115_5E201_RY601_CV(bPortKNX := 1, dwIndex_DPT := 115, typDPT := typDPT);
STLV80_563.STLV80_A_563_5E201.RY601_CV := M1_115_5E201_RY601_CV.rValue_OUT;
(* LH601_OP *)
(* LH601_CMD *)
M1_116_5E201_LH601_OP(bPortKNX := 1, dwIndex_DPT := 116, rValue_IN := STLV80_563.STLV80_A_563_5E201.LH601_OP, xUpdate_KNX := i = 40, typDPT := typDPT);
M1_117_5E201_LH601_CMD(bPortKNX := 1, dwIndex_DPT := 117, xSwitch_IN := STLV80_563.STLV80_A_563_5E201.LH601_CMD, xUpdate_KNX := i = 41, typDPT := typDPT);
(* LC601_OP *)
(* LC602_OP *)
M1_118_5E201_LC601_OP(bPortKNX := 1, dwIndex_DPT := 118, rValue_IN := STLV80_563.STLV80_A_563_5E201.LC601_OP, xUpdate_KNX := i = 42, typDPT := typDPT);
M1_119_5E201_LC602_OP(bPortKNX := 1, dwIndex_DPT := 119, rValue_IN := STLV80_563.STLV80_A_563_5E201.LC602_OP, xUpdate_KNX := i = 43, typDPT := typDPT);
(* LC601_CMD *)
(* RT601_SP *)
M1_120_5E201_LC601_CMD(bPortKNX := 1, dwIndex_DPT := 120, xSwitch_IN := STLV80_563.STLV80_A_563_5E201.LC601_CMD, xUpdate_KNX := i = 44, typDPT := typDPT);
M1_121_5E201_RT601_SP(bPortKNX := 1, dwIndex_DPT := 121, rValue_IN := STLV80_563.STLV80_A_563_5E201.RT601_SP_D, xUpdate_KNX := NOT STLV80_563.STLV80_A_563_5E201.RB601_HVAC, typDPT := typDPT);
(* RT601_SP Feedback *)
M1_122_5E201_RT601_SP_FB(bPortKNX := 1, dwIndex_DPT := 122, typDPT := typDPT);
STLV80_563.STLV80_A_563_5E201.RT601_SP_IN := M1_122_5E201_RT601_SP_FB.rValue_OUT;
(* Rom 5E202 *)
(* RB601_V *)
(* RB601_HVAC *)
M1_123_5E202_RB601_V(bPortKNX := 1, dwIndex_DPT := 123, typDPT := typDPT);
STLV80_563.STLV80_A_563_5E202.RB601_V := M1_123_5E202_RB601_V.xSwitch_OUT;
M1_124_5E202_RB601_HVAC(bPortKNX := 1, dwIndex_DPT := 124, typDPT := typDPT);
STLV80_563.STLV80_A_563_5E202.RB601_HVAC := M1_124_5E202_RB601_HVAC.xSwitch_OUT;
(* RT601_CT *)
(* RY601_CV *)
M1_125_5E202_RT601_CT(bPortKNX := 1, dwIndex_DPT := 125, typDPT := typDPT);
STLV80_563.STLV80_A_563_5E202.RT601_CT := M1_125_5E202_RT601_CT.rValue_OUT;
M1_126_5E202_RY601_CV(bPortKNX := 1, dwIndex_DPT := 126, typDPT := typDPT);
STLV80_563.STLV80_A_563_5E202.RY601_CV := M1_126_5E202_RY601_CV.rValue_OUT;
(* LH601_OP *)
(* LH601_CMD *)
M1_127_5E202_LH601_OP(bPortKNX := 1, dwIndex_DPT := 127, rValue_IN := STLV80_563.STLV80_A_563_5E202.LH601_OP, xUpdate_KNX := i = 45, typDPT := typDPT);
M1_128_5E202_LH601_CMD(bPortKNX := 1, dwIndex_DPT := 128, xSwitch_IN := STLV80_563.STLV80_A_563_5E202.LH601_CMD, xUpdate_KNX := i = 46, typDPT := typDPT);
(* LC601_OP *)
(* LC601_CMD *)
M1_129_5E202_LC601_OP(bPortKNX := 1, dwIndex_DPT := 129, rValue_IN := STLV80_563.STLV80_A_563_5E202.LC601_OP, xUpdate_KNX := i = 47, typDPT := typDPT);
M1_130_5E202_LC601_CMD(bPortKNX := 1, dwIndex_DPT := 130, xSwitch_IN := STLV80_563.STLV80_A_563_5E202.LC601_CMD, xUpdate_KNX := i = 48, typDPT := typDPT);
(* LC602_CMD *)
(* RT601_SP *)
M1_131_5E202_LC602_CMD(bPortKNX := 1, dwIndex_DPT := 131, xSwitch_IN := STLV80_563.STLV80_A_563_5E202.LC602_CMD, xUpdate_KNX := i = 49, typDPT := typDPT);
M1_132_5E202_RT601_SP(bPortKNX := 1, dwIndex_DPT := 132, rValue_IN := STLV80_563.STLV80_A_563_5E202.RT601_SP_D, xUpdate_KNX := NOT STLV80_563.STLV80_A_563_5E202.RB601_HVAC, typDPT := typDPT);
(* RT601_SP Feedback *)
M1_133_5E202_RT601_SP_FB(bPortKNX := 1, dwIndex_DPT := 133, typDPT := typDPT);
STLV80_563.STLV80_A_563_5E202.RT601_SP_IN := M1_133_5E202_RT601_SP_FB.rValue_OUT;
(* Rom 5E301 *)
(* RB601_V *)
(* RB601_HVAC *)
M1_134_5E301_RB601_V(bPortKNX := 1, dwIndex_DPT := 134, typDPT := typDPT);
STLV80_563.STLV80_A_563_5E301.RB601_V := M1_134_5E301_RB601_V.xSwitch_OUT;
M1_135_5E301_RB601_HVAC(bPortKNX := 1, dwIndex_DPT := 135, typDPT := typDPT);
STLV80_563.STLV80_A_563_5E301.RB601_HVAC := M1_135_5E301_RB601_HVAC.xSwitch_OUT;
(* RT601_CT *)
(* RT602_CT *)
M1_136_5E301_RT601_CT(bPortKNX := 1, dwIndex_DPT := 136, typDPT := typDPT);
STLV80_563.STLV80_A_563_5E301.RT601_CT := M1_136_5E301_RT601_CT.rValue_OUT;
M1_137_5E301_RT602_CT(bPortKNX := 1, dwIndex_DPT := 137, typDPT := typDPT);
STLV80_563.STLV80_A_563_5E301.RT602_CT := M1_137_5E301_RT602_CT.rValue_OUT;
(* RY601_CV *)
(* LH601_OP *)
M1_138_5E301_RY601_CV(bPortKNX := 1, dwIndex_DPT := 138, typDPT := typDPT);
STLV80_563.STLV80_A_563_5E301.RY601_CV := M1_138_5E301_RY601_CV.rValue_OUT;
M1_139_5E301_LH601_OP(bPortKNX := 1, dwIndex_DPT := 139, rValue_IN := STLV80_563.STLV80_A_563_5E301.LH601_OP, xUpdate_KNX := i = 50, typDPT := typDPT);
(* LH601_CMD *)
(* LC601_OP *)
M1_140_5E301_LH601_CMD(bPortKNX := 1, dwIndex_DPT := 140, xSwitch_IN := STLV80_563.STLV80_A_563_5E301.LH601_CMD, xUpdate_KNX := i = 51, typDPT := typDPT);
M1_141_5E301_LC601_OP(bPortKNX := 1, dwIndex_DPT := 141, rValue_IN := STLV80_563.STLV80_A_563_5E301.LC601_OP, xUpdate_KNX := i = 52, typDPT := typDPT);
(* LC601_CMD *)
(* RT601_SP *)
M1_142_5E301_LC601_CMD(bPortKNX := 1, dwIndex_DPT := 142, xSwitch_IN := STLV80_563.STLV80_A_563_5E301.LC601_CMD, xUpdate_KNX := i = 53, typDPT := typDPT);
M1_143_5E301_RT601_SP(bPortKNX := 1, dwIndex_DPT := 143, rValue_IN := STLV80_563.STLV80_A_563_5E301.RT601_SP_D, xUpdate_KNX := NOT STLV80_563.STLV80_A_563_5E301.RB601_HVAC, typDPT := typDPT);
(* RT602_SP *)
(* RT601_SP Feedback *)
M1_144_5E301_RT602_SP(bPortKNX := 1, dwIndex_DPT := 144, rValue_IN := STLV80_563.STLV80_A_563_5E301.RT602_SP, xUpdate_KNX := NOT STLV80_563.STLV80_A_563_5E301.RB601_HVAC, typDPT := typDPT);
M1_145_5E301_RT601_SP_FB(bPortKNX := 1, dwIndex_DPT := 145, typDPT := typDPT);
STLV80_563.STLV80_A_563_5E301.RT601_SP_IN := M1_145_5E301_RT601_SP_FB.rValue_OUT;
(* Rom 5E302 *)
(* RB601_V *)
(* RB601_HVAC *)
M1_146_5E302_RB601_V(bPortKNX := 1, dwIndex_DPT := 146, typDPT := typDPT);
STLV80_563.STLV80_A_563_5E302.RB601_V := M1_146_5E302_RB601_V.xSwitch_OUT;
M1_147_5E302_RB601_HVAC(bPortKNX := 1, dwIndex_DPT := 147, typDPT := typDPT);
STLV80_563.STLV80_A_563_5E302.RB601_HVAC := M1_147_5E302_RB601_HVAC.xSwitch_OUT;
(* RT601_CT *)
(* RY601_CV *)
M1_148_5E302_RT601_CT(bPortKNX := 1, dwIndex_DPT := 148, typDPT := typDPT);
STLV80_563.STLV80_A_563_5E302.RT601_CT := M1_148_5E302_RT601_CT.rValue_OUT;
M1_149_5E302_RY601_CV(bPortKNX := 1, dwIndex_DPT := 149, typDPT := typDPT);
STLV80_563.STLV80_A_563_5E302.RY601_CV := M1_149_5E302_RY601_CV.rValue_OUT;
(* LH601_OP *)
(* LH601_CMD *)
M1_150_5E302_LH601_OP(bPortKNX := 1, dwIndex_DPT := 150, rValue_IN := STLV80_563.STLV80_A_563_5E302.LH601_OP, xUpdate_KNX := i = 54, typDPT := typDPT);
M1_151_5E302_LH601_CMD(bPortKNX := 1, dwIndex_DPT := 151, xSwitch_IN := STLV80_563.STLV80_A_563_5E302.LH601_CMD, xUpdate_KNX := i = 55, typDPT := typDPT);
(* LC601_OP *)
(* LC601_CMD *)
M1_152_5E302_LC601_OP(bPortKNX := 1, dwIndex_DPT := 152, rValue_IN := STLV80_563.STLV80_A_563_5E302.LC601_OP, xUpdate_KNX := i = 56, typDPT := typDPT);
M1_153_5E302_LC601_CMD(bPortKNX := 1, dwIndex_DPT := 153, xSwitch_IN := STLV80_563.STLV80_A_563_5E302.LC601_CMD, xUpdate_KNX := i = 57, typDPT := typDPT);
(* RT601_SP *)
(* RT601_SP Feedback *)
M1_154_5E302_RT601_SP(bPortKNX := 1, dwIndex_DPT := 154, rValue_IN := STLV80_563.STLV80_A_563_5E302.RT601_SP_D, xUpdate_KNX := NOT STLV80_563.STLV80_A_563_5E302.RB601_HVAC, typDPT := typDPT);
M1_155_5E302_RT601_SP_FB(bPortKNX := 1, dwIndex_DPT := 155, typDPT := typDPT);
STLV80_563.STLV80_A_563_5E302.RT601_SP_IN := M1_155_5E302_RT601_SP_FB.rValue_OUT;
(* RT602_SP Feedback *)
M1_156_5E302_RT602_SP_FB(bPortKNX := 1, dwIndex_DPT := 156, typDPT := typDPT);
STLV80_563.STLV80_A_563_5E302.RT602_SP_IN := M1_156_5E302_RT602_SP_FB.rValue_OUT;
(* Rom 5F201 *)
(* RB601_V *)
(* RB602_V *)
M1_157_5F201_RB601_V(bPortKNX := 1, dwIndex_DPT := 157, typDPT := typDPT);
STLV80_563.STLV80_A_563_5F201.RB601_V := M1_157_5F201_RB601_V.xSwitch_OUT;
M1_158_5F201_RB602_V(bPortKNX := 1, dwIndex_DPT := 158, typDPT := typDPT);
STLV80_563.STLV80_A_563_5F201.RB602_V := M1_158_5F201_RB602_V.xSwitch_OUT;
(* RB603_V *)
(* RB604_V *)
M1_159_5F201_RB603_V(bPortKNX := 1, dwIndex_DPT := 159, typDPT := typDPT);
STLV80_563.STLV80_A_563_5F201.RB603_V := M1_159_5F201_RB603_V.xSwitch_OUT;
M1_160_5F201_RB604_V(bPortKNX := 1, dwIndex_DPT := 160, typDPT := typDPT);
STLV80_563.STLV80_A_563_5F201.RB604_V := M1_160_5F201_RB604_V.xSwitch_OUT;
(* RB601_HVAC *)
(* RT601_CT *)
M1_161_5F201_RB601_HVAC(bPortKNX := 1, dwIndex_DPT := 161, typDPT := typDPT);
STLV80_563.STLV80_A_563_5F201.RB601_HVAC := M1_161_5F201_RB601_HVAC.xSwitch_OUT;
M1_162_5F201_RT601_CT(bPortKNX := 1, dwIndex_DPT := 162, typDPT := typDPT);
STLV80_563.STLV80_A_563_5F201.RT601_CT := M1_162_5F201_RT601_CT.rValue_OUT;
(* RY601_CV *)
(* LH601_OP *)
M1_163_5F201_RY601_CV(bPortKNX := 1, dwIndex_DPT := 163, typDPT := typDPT);
STLV80_563.STLV80_A_563_5F201.RY601_CV := M1_163_5F201_RY601_CV.rValue_OUT;
M1_164_5F201_LH601_OP(bPortKNX := 1, dwIndex_DPT := 164, rValue_IN := STLV80_563.STLV80_A_563_5F201.LH601_OP, xUpdate_KNX := i = 58, typDPT := typDPT);
(* LH601_CMD *)
(* LC601_OP *)
M1_165_5F201_LH601_CMD(bPortKNX := 1, dwIndex_DPT := 165, xSwitch_IN := STLV80_563.STLV80_A_563_5F201.LH601_CMD, xUpdate_KNX := i = 59, typDPT := typDPT);
M1_166_5F201_LC601_OP(bPortKNX := 1, dwIndex_DPT := 166, rValue_IN := STLV80_563.STLV80_A_563_5F201.LC601_OP, xUpdate_KNX := i = 60, typDPT := typDPT);
(* LC601_CMD *)
(* RT601_SP *)
M1_167_5F201_LC601_CMD(bPortKNX := 1, dwIndex_DPT := 167, xSwitch_IN := STLV80_563.STLV80_A_563_5F201.LC601_CMD, xUpdate_KNX := i = 61, typDPT := typDPT);
M1_168_5F201_RT601_SP(bPortKNX := 1, dwIndex_DPT := 168, rValue_IN := STLV80_563.STLV80_A_563_5F201.RT601_SP_D, xUpdate_KNX := NOT STLV80_563.STLV80_A_563_5F201.RB601_HVAC, typDPT := typDPT);
(* RT601_SP Feedback *)
M1_169_5F201_RT601_SP_FB(bPortKNX := 1, dwIndex_DPT := 169, typDPT := typDPT);
STLV80_563.STLV80_A_563_5F201.RT601_SP_IN := M1_169_5F201_RT601_SP_FB.rValue_OUT;
(* Rom 5F202 *)
(* RB601_V *)
(* RB602_V *)
M1_170_5F202_RB601_V(bPortKNX := 1, dwIndex_DPT := 170, typDPT := typDPT);
STLV80_563.STLV80_A_563_5F202.RB601_V := M1_170_5F202_RB601_V.xSwitch_OUT;
M1_171_5F202_RB602_V(bPortKNX := 1, dwIndex_DPT := 171, typDPT := typDPT);
STLV80_563.STLV80_A_563_5F202.RB602_V := M1_171_5F202_RB602_V.xSwitch_OUT;
(* RB603_V *)
(* RB604_V *)
M1_172_5F202_RB603_V(bPortKNX := 1, dwIndex_DPT := 172, typDPT := typDPT);
STLV80_563.STLV80_A_563_5F202.RB603_V := M1_172_5F202_RB603_V.xSwitch_OUT;
M1_173_5F202_RB604_V(bPortKNX := 1, dwIndex_DPT := 173, typDPT := typDPT);
STLV80_563.STLV80_A_563_5F202.RB604_V := M1_173_5F202_RB604_V.xSwitch_OUT;
(* RB605_V *)
(* RB601_HVAC *)
M1_174_5F202_RB605_V(bPortKNX := 1, dwIndex_DPT := 174, typDPT := typDPT);
STLV80_563.STLV80_A_563_5F202.RB605_V := M1_174_5F202_RB605_V.xSwitch_OUT;
M1_175_5F202_RB601_HVAC(bPortKNX := 1, dwIndex_DPT := 175, typDPT := typDPT);
STLV80_563.STLV80_A_563_5F202.RB601_HVAC := M1_175_5F202_RB601_HVAC.xSwitch_OUT;
(* RB602_HVAC *)
(* RB603_HVAC *)
M1_176_5F202_RB602_HVAC(bPortKNX := 1, dwIndex_DPT := 176, typDPT := typDPT);
STLV80_563.STLV80_A_563_5F202.RB602_HVAC := M1_176_5F202_RB602_HVAC.xSwitch_OUT;
M1_177_5F202_RB603_HVAC(bPortKNX := 1, dwIndex_DPT := 177, typDPT := typDPT);
STLV80_563.STLV80_A_563_5F202.RB603_HVAC := M1_177_5F202_RB603_HVAC.xSwitch_OUT;
(* RB604_HVAC *)
(* RB605_HVAC *)
M1_178_5F202_RB604_HVAC(bPortKNX := 1, dwIndex_DPT := 178, typDPT := typDPT);
STLV80_563.STLV80_A_563_5F202.RB604_HVAC := M1_178_5F202_RB604_HVAC.xSwitch_OUT;
M1_179_5F202_RB605_HVAC(bPortKNX := 1, dwIndex_DPT := 179, typDPT := typDPT);
STLV80_563.STLV80_A_563_5F202.RB605_HVAC := M1_179_5F202_RB605_HVAC.xSwitch_OUT;
(* RT601_CT *)
(* RT602_CT *)
M1_180_5F202_RT601_CT(bPortKNX := 1, dwIndex_DPT := 180, typDPT := typDPT);
STLV80_563.STLV80_A_563_5F202.RT601_CT := M1_180_5F202_RT601_CT.rValue_OUT;
M1_181_5F202_RT602_CT(bPortKNX := 1, dwIndex_DPT := 181, typDPT := typDPT);
STLV80_563.STLV80_A_563_5F202.RT602_CT := M1_181_5F202_RT602_CT.rValue_OUT;
(* RY601_CV *)
(* LH601_OP *)
M1_182_5F202_RY601_CV(bPortKNX := 1, dwIndex_DPT := 182, typDPT := typDPT);
STLV80_563.STLV80_A_563_5F202.RY601_CV := M1_182_5F202_RY601_CV.rValue_OUT;
M1_183_5F202_LH601_OP(bPortKNX := 1, dwIndex_DPT := 183, rValue_IN := STLV80_563.STLV80_A_563_5F202.LH601_OP, xUpdate_KNX := i = 62, typDPT := typDPT);
(* LH601_CMD *)
(* LC601_OP *)
M1_184_5F202_LH601_CMD(bPortKNX := 1, dwIndex_DPT := 184, xSwitch_IN := STLV80_563.STLV80_A_563_5F202.LH601_CMD, xUpdate_KNX := i = 63, typDPT := typDPT);
M1_185_5F202_LC601_OP(bPortKNX := 1, dwIndex_DPT := 185, rValue_IN := STLV80_563.STLV80_A_563_5F202.LC601_OP, xUpdate_KNX := i = 64, typDPT := typDPT);
(* LC601_CMD *)
(* RT601_SP *)
M1_186_5F202_LC601_CMD(bPortKNX := 1, dwIndex_DPT := 186, xSwitch_IN := STLV80_563.STLV80_A_563_5F202.LC601_CMD, xUpdate_KNX := i = 65, typDPT := typDPT);
M1_187_5F202_RT601_SP(bPortKNX := 1, dwIndex_DPT := 187, rValue_IN := STLV80_563.STLV80_A_563_5F202.RT601_SP_D, xUpdate_KNX := NOT STLV80_563.STLV80_A_563_5F202.RB601_HVAC, typDPT := typDPT);
(* RT601_SP Feedback *)
M1_188_5F202_RT601_SP_FB(bPortKNX := 1, dwIndex_DPT := 188, typDPT := typDPT);
STLV80_563.STLV80_A_563_5F202.RT601_SP_IN := M1_188_5F202_RT601_SP_FB.rValue_OUT;
(* Rom 5F301 *)
(* RB601_V *)
(* RB601_HVAC *)
M1_189_5F301_RB601_V(bPortKNX := 1, dwIndex_DPT := 189, typDPT := typDPT);
STLV80_563.STLV80_A_563_5F301.RB601_V := M1_189_5F301_RB601_V.xSwitch_OUT;
M1_190_5F301_RB601_HVAC(bPortKNX := 1, dwIndex_DPT := 190, typDPT := typDPT);
STLV80_563.STLV80_A_563_5F301.RB601_HVAC := M1_190_5F301_RB601_HVAC.xSwitch_OUT;
(* RT601_CT *)
(* RY601_CV *)
M1_191_5F301_RT601_CT(bPortKNX := 1, dwIndex_DPT := 191, typDPT := typDPT);
STLV80_563.STLV80_A_563_5F301.RT601_CT := M1_191_5F301_RT601_CT.rValue_OUT;
M1_192_5F301_RY601_CV(bPortKNX := 1, dwIndex_DPT := 192, typDPT := typDPT);
STLV80_563.STLV80_A_563_5F301.RY601_CV := M1_192_5F301_RY601_CV.rValue_OUT;
(* LH601_OP *)
(* LH601_CMD *)
M1_193_5F301_LH601_OP(bPortKNX := 1, dwIndex_DPT := 193, rValue_IN := STLV80_563.STLV80_A_563_5F301.LH601_OP, xUpdate_KNX := i = 66, typDPT := typDPT);
M1_194_5F301_LH601_CMD(bPortKNX := 1, dwIndex_DPT := 194, xSwitch_IN := STLV80_563.STLV80_A_563_5F301.LH601_CMD, xUpdate_KNX := i = 67, typDPT := typDPT);
(* LC601_OP *)
(* LC601_CMD *)
M1_195_5F301_LC601_OP(bPortKNX := 1, dwIndex_DPT := 195, rValue_IN := STLV80_563.STLV80_A_563_5F301.LC601_OP, xUpdate_KNX := i = 68, typDPT := typDPT);
M1_196_5F301_LC601_CMD(bPortKNX := 1, dwIndex_DPT := 196, xSwitch_IN := STLV80_563.STLV80_A_563_5F301.LC601_CMD, xUpdate_KNX := i = 69, typDPT := typDPT);
(* RT601_SP *)
(* RT601_SP Feedback *)
M1_197_5F301_RT601_SP(bPortKNX := 1, dwIndex_DPT := 197, rValue_IN := STLV80_563.STLV80_A_563_5F301.RT601_SP_D, xUpdate_KNX := NOT STLV80_563.STLV80_A_563_5F301.RB601_HVAC, typDPT := typDPT);
M1_198_5F301_RT601_SP_FB(bPortKNX := 1, dwIndex_DPT := 198, typDPT := typDPT);
STLV80_563.STLV80_A_563_5F301.RT601_SP_IN := M1_198_5F301_RT601_SP_FB.rValue_OUT;
(* Rom 5F302 *)
(* RB601_V *)
(* RB601_HVAC *)
M1_199_5F302_RB601_V(bPortKNX := 1, dwIndex_DPT := 199, typDPT := typDPT);
STLV80_563.STLV80_A_563_5F302.RB601_V := M1_199_5F302_RB601_V.xSwitch_OUT;
M1_200_5F302_RB601_HVAC(bPortKNX := 1, dwIndex_DPT := 200, typDPT := typDPT);
STLV80_563.STLV80_A_563_5F302.RB601_HVAC := M1_200_5F302_RB601_HVAC.xSwitch_OUT;
(* RT601_CT *)
(* RY601_CV *)
M1_201_5F302_RT601_CT(bPortKNX := 1, dwIndex_DPT := 201, typDPT := typDPT);
STLV80_563.STLV80_A_563_5F302.RT601_CT := M1_201_5F302_RT601_CT.rValue_OUT;
M1_202_5F302_RY601_CV(bPortKNX := 1, dwIndex_DPT := 202, typDPT := typDPT);
STLV80_563.STLV80_A_563_5F302.RY601_CV := M1_202_5F302_RY601_CV.rValue_OUT;
(* LH601_OP *)
(* LH601_CMD *)
M1_203_5F302_LH601_OP(bPortKNX := 1, dwIndex_DPT := 203, rValue_IN := STLV80_563.STLV80_A_563_5F302.LH601_OP, xUpdate_KNX := i = 70, typDPT := typDPT);
M1_204_5F302_LH601_CMD(bPortKNX := 1, dwIndex_DPT := 204, xSwitch_IN := STLV80_563.STLV80_A_563_5F302.LH601_CMD, xUpdate_KNX := i = 71, typDPT := typDPT);
(* LC601_OP *)
(* LC601_CMD *)
M1_205_5F302_LC601_OP(bPortKNX := 1, dwIndex_DPT := 205, rValue_IN := STLV80_563.STLV80_A_563_5F302.LC601_OP, xUpdate_KNX := i = 72, typDPT := typDPT);
M1_206_5F302_LC601_CMD(bPortKNX := 1, dwIndex_DPT := 206, xSwitch_IN := STLV80_563.STLV80_A_563_5F302.LC601_CMD, xUpdate_KNX := i = 73, typDPT := typDPT);
(* RT601_SP *)
(* RT601_SP Feedback *)
M1_207_5F302_RT601_SP(bPortKNX := 1, dwIndex_DPT := 207, rValue_IN := STLV80_563.STLV80_A_563_5F302.RT601_SP_D, xUpdate_KNX := NOT STLV80_563.STLV80_A_563_5F302.RB601_HVAC, typDPT := typDPT);
M1_208_5F302_RT601_SP_FB(bPortKNX := 1, dwIndex_DPT := 208, typDPT := typDPT);
STLV80_563.STLV80_A_563_5F302.RT601_SP_IN := M1_208_5F302_RT601_SP_FB.rValue_OUT;
(* Rom 5G201 *)
(* RB601_V *)
(* RB601_HVAC *)
M1_209_5G201_RB601_V(bPortKNX := 1, dwIndex_DPT := 209, typDPT := typDPT);
STLV80_563.STLV80_A_563_5G201.RB601_V := M1_209_5G201_RB601_V.xSwitch_OUT;
M1_210_5G201_RB601_HVAC(bPortKNX := 1, dwIndex_DPT := 210, typDPT := typDPT);
STLV80_563.STLV80_A_563_5G201.RB601_HVAC := M1_210_5G201_RB601_HVAC.xSwitch_OUT;
(* RT601_CT *)
(* RY601_CV *)
M1_211_5G201_RT601_CT(bPortKNX := 1, dwIndex_DPT := 211, typDPT := typDPT);
STLV80_563.STLV80_A_563_5G201.RT601_CT := M1_211_5G201_RT601_CT.rValue_OUT;
M1_212_5G201_RY601_CV(bPortKNX := 1, dwIndex_DPT := 212, typDPT := typDPT);
STLV80_563.STLV80_A_563_5G201.RY601_CV := M1_212_5G201_RY601_CV.rValue_OUT;
(* LH601_OP *)
(* LH601_CMD *)
M1_213_5G201_LH601_OP(bPortKNX := 1, dwIndex_DPT := 213, rValue_IN := STLV80_563.STLV80_A_563_5G201.LH601_OP, xUpdate_KNX := i = 74, typDPT := typDPT);
M1_214_5G201_LH601_CMD(bPortKNX := 1, dwIndex_DPT := 214, xSwitch_IN := STLV80_563.STLV80_A_563_5G201.LH601_CMD, xUpdate_KNX := i = 75, typDPT := typDPT);
(* LC601_OP *)
(* LC601_CMD *)
M1_215_5G201_LC601_OP(bPortKNX := 1, dwIndex_DPT := 215, rValue_IN := STLV80_563.STLV80_A_563_5G201.LC601_OP, xUpdate_KNX := i = 76, typDPT := typDPT);
M1_216_5G201_LC601_CMD(bPortKNX := 1, dwIndex_DPT := 216, xSwitch_IN := STLV80_563.STLV80_A_563_5G201.LC601_CMD, xUpdate_KNX := i = 77, typDPT := typDPT);
(* RT601_SP *)
(* RT601_SP Feedback *)
M1_217_5G201_RT601_SP(bPortKNX := 1, dwIndex_DPT := 217, rValue_IN := STLV80_563.STLV80_A_563_5G201.RT601_SP_D, xUpdate_KNX := NOT STLV80_563.STLV80_A_563_5G201.RB601_HVAC, typDPT := typDPT);
M1_218_5G201_RT601_SP_FB(bPortKNX := 1, dwIndex_DPT := 218, typDPT := typDPT);
STLV80_563.STLV80_A_563_5G201.RT601_SP_IN := M1_218_5G201_RT601_SP_FB.rValue_OUT;
(* Rom 5G202 *)
(* RB601_V *)
(* RB601_HVAC *)
M1_219_5G202_RB601_V(bPortKNX := 1, dwIndex_DPT := 219, typDPT := typDPT);
STLV80_563.STLV80_A_563_5G202.RB601_V := M1_219_5G202_RB601_V.xSwitch_OUT;
M1_220_5G202_RB601_HVAC(bPortKNX := 1, dwIndex_DPT := 220, typDPT := typDPT);
STLV80_563.STLV80_A_563_5G202.RB601_HVAC := M1_220_5G202_RB601_HVAC.xSwitch_OUT;
(* RT601_CT *)
(* RY601_CV *)
M1_221_5G202_RT601_CT(bPortKNX := 1, dwIndex_DPT := 221, typDPT := typDPT);
STLV80_563.STLV80_A_563_5G202.RT601_CT := M1_221_5G202_RT601_CT.rValue_OUT;
M1_222_5G202_RY601_CV(bPortKNX := 1, dwIndex_DPT := 222, typDPT := typDPT);
STLV80_563.STLV80_A_563_5G202.RY601_CV := M1_222_5G202_RY601_CV.rValue_OUT;
(* LH601_OP *)
(* LH601_CMD *)
M1_223_5G202_LH601_OP(bPortKNX := 1, dwIndex_DPT := 223, rValue_IN := STLV80_563.STLV80_A_563_5G202.LH601_OP, xUpdate_KNX := i = 78, typDPT := typDPT);
M1_224_5G202_LH601_CMD(bPortKNX := 1, dwIndex_DPT := 224, xSwitch_IN := STLV80_563.STLV80_A_563_5G202.LH601_CMD, xUpdate_KNX := i = 79, typDPT := typDPT);
(* LC601_OP *)
(* LC601_CMD *)
M1_225_5G202_LC601_OP(bPortKNX := 1, dwIndex_DPT := 225, rValue_IN := STLV80_563.STLV80_A_563_5G202.LC601_OP, xUpdate_KNX := i = 80, typDPT := typDPT);
M1_226_5G202_LC601_CMD(bPortKNX := 1, dwIndex_DPT := 226, xSwitch_IN := STLV80_563.STLV80_A_563_5G202.LC601_CMD, xUpdate_KNX := i = 81, typDPT := typDPT);
(* RT601_SP *)
(* RT601_SP Feedback *)
M1_227_5G202_RT601_SP(bPortKNX := 1, dwIndex_DPT := 227, rValue_IN := STLV80_563.STLV80_A_563_5G202.RT601_SP_D, xUpdate_KNX := NOT STLV80_563.STLV80_A_563_5G202.RB601_HVAC, typDPT := typDPT);
M1_228_5G202_RT601_SP_FB(bPortKNX := 1, dwIndex_DPT := 228, typDPT := typDPT);
STLV80_563.STLV80_A_563_5G202.RT601_SP_IN := M1_228_5G202_RT601_SP_FB.rValue_OUT;
(* Rom 5H301 *)
(* RB601_V *)
(* RB601_HVAC *)
M1_229_5H301_RB601_V(bPortKNX := 1, dwIndex_DPT := 229, typDPT := typDPT);
STLV80_563.STLV80_A_563_5H301.RB601_V := M1_229_5H301_RB601_V.xSwitch_OUT;
M1_230_5H301_RB601_HVAC(bPortKNX := 1, dwIndex_DPT := 230, typDPT := typDPT);
STLV80_563.STLV80_A_563_5H301.RB601_HVAC := M1_230_5H301_RB601_HVAC.xSwitch_OUT;
(* RT601_CT *)
(* RY601_CV *)
M1_231_5H301_RT601_CT(bPortKNX := 1, dwIndex_DPT := 231, typDPT := typDPT);
STLV80_563.STLV80_A_563_5H301.RT601_CT := M1_231_5H301_RT601_CT.rValue_OUT;
M1_232_5H301_RY601_CV(bPortKNX := 1, dwIndex_DPT := 232, typDPT := typDPT);
STLV80_563.STLV80_A_563_5H301.RY601_CV := M1_232_5H301_RY601_CV.rValue_OUT;
(* LH601_OP *)
(* LH601_CMD *)
M1_233_5H301_LH601_OP(bPortKNX := 1, dwIndex_DPT := 233, rValue_IN := STLV80_563.STLV80_A_563_5H301.LH601_OP, xUpdate_KNX := i = 82, typDPT := typDPT);
M1_234_5H301_LH601_CMD(bPortKNX := 1, dwIndex_DPT := 234, xSwitch_IN := STLV80_563.STLV80_A_563_5H301.LH601_CMD, xUpdate_KNX := i = 83, typDPT := typDPT);
(* LC601_OP *)
(* LC601_CMD *)
M1_235_5H301_LC601_OP(bPortKNX := 1, dwIndex_DPT := 235, rValue_IN := STLV80_563.STLV80_A_563_5H301.LC601_OP, xUpdate_KNX := i = 84, typDPT := typDPT);
M1_236_5H301_LC601_CMD(bPortKNX := 1, dwIndex_DPT := 236, xSwitch_IN := STLV80_563.STLV80_A_563_5H301.LC601_CMD, xUpdate_KNX := i = 85, typDPT := typDPT);
(* RT601_SP *)
(* RT601_SP Feedback *)
M1_237_5H301_RT601_SP(bPortKNX := 1, dwIndex_DPT := 237, rValue_IN := STLV80_563.STLV80_A_563_5H301.RT601_SP_D, xUpdate_KNX := NOT STLV80_563.STLV80_A_563_5H301.RB601_HVAC, typDPT := typDPT);
M1_238_5H301_RT601_SP_FB(bPortKNX := 1, dwIndex_DPT := 238, typDPT := typDPT);
STLV80_563.STLV80_A_563_5H301.RT601_SP_IN := M1_238_5H301_RT601_SP_FB.rValue_OUT;
(* Rom 5H302 *)
(* RB601_V *)
(* RB601_HVAC *)
M1_239_5H302_RB601_V(bPortKNX := 1, dwIndex_DPT := 239, typDPT := typDPT);
STLV80_563.STLV80_A_563_5H302.RB601_V := M1_239_5H302_RB601_V.xSwitch_OUT;
M1_240_5H302_RB601_HVAC(bPortKNX := 1, dwIndex_DPT := 240, typDPT := typDPT);
STLV80_563.STLV80_A_563_5H302.RB601_HVAC := M1_240_5H302_RB601_HVAC.xSwitch_OUT;
(* RT601_CT *)
(* RY601_CV *)
M1_241_5H302_RT601_CT(bPortKNX := 1, dwIndex_DPT := 241, typDPT := typDPT);
STLV80_563.STLV80_A_563_5H302.RT601_CT := M1_241_5H302_RT601_CT.rValue_OUT;
M1_242_5H302_RY601_CV(bPortKNX := 1, dwIndex_DPT := 242, typDPT := typDPT);
STLV80_563.STLV80_A_563_5H302.RY601_CV := M1_242_5H302_RY601_CV.rValue_OUT;
(* LH601_OP *)
(* LH601_CMD *)
M1_243_5H302_LH601_OP(bPortKNX := 1, dwIndex_DPT := 243, rValue_IN := STLV80_563.STLV80_A_563_5H302.LH601_OP, xUpdate_KNX := i = 86, typDPT := typDPT);
M1_244_5H302_LH601_CMD(bPortKNX := 1, dwIndex_DPT := 244, xSwitch_IN := STLV80_563.STLV80_A_563_5H302.LH601_CMD, xUpdate_KNX := i = 87, typDPT := typDPT);
(* LC601_OP *)
(* LC601_CMD *)
M1_245_5H302_LC601_OP(bPortKNX := 1, dwIndex_DPT := 245, rValue_IN := STLV80_563.STLV80_A_563_5H302.LC601_OP, xUpdate_KNX := i = 88, typDPT := typDPT);
M1_246_5H302_LC601_CMD(bPortKNX := 1, dwIndex_DPT := 246, xSwitch_IN := STLV80_563.STLV80_A_563_5H302.LC601_CMD, xUpdate_KNX := i = 89, typDPT := typDPT);
(* RT601_SP *)
(* RT601_SP Feedback *)
M1_247_5H302_RT601_SP(bPortKNX := 1, dwIndex_DPT := 247, rValue_IN := STLV80_563.STLV80_A_563_5H302.RT601_SP_D, xUpdate_KNX := NOT STLV80_563.STLV80_A_563_5H302.RB601_HVAC, typDPT := typDPT);
M1_248_5H302_RT601_SP_FB(bPortKNX := 1, dwIndex_DPT := 248, typDPT := typDPT);
STLV80_563.STLV80_A_563_5H302.RT601_SP_IN := M1_248_5H302_RT601_SP_FB.rValue_OUT;
END_PROGRAM

PROGRAM PRG_563_KNX_2
  VAR
    i : INT := 0;  (* Felles *)
    Interval : OSCAT_BASIC.CLK_PRG;
    typDPT : typDPT;
    KNX_master_2 : WagoAppKNX.FbKNX_Master;  (* Master *)
    M2_001_5H201_RB601_V : fbDPT_Switch_pro;  (* 5H201 *)
    M2_002_5H201_RB601_HVAC : fbDPT_Switch_pro;
    M2_003_5H201_RT601_CT : fbDPT_Value_Temp_pro;
    M2_004_5H201_RY601_CV : fbDPT_Value_AirQuality_pro;
    M2_005_5H201_LH601_OP : fbDPT_Scaling_pro;
    M2_006_5H201_LH601_CMD : fbDPT_Switch_pro;
    M2_007_5H201_LC601_OP : fbDPT_Scaling_pro;
    M2_008_5H201_LC601_CMD : fbDPT_Switch_pro;
    M2_009_5H201_RT601_SP : fbDPT_Value_Temp_pro;
    M2_010_5H201_RT601_SP_FB : fbDPT_Value_Temp_pro;
    M2_011_5I202_RB601_V : fbDPT_Switch_pro;  (* 5I202 *)
    M2_012_5I202_RB601_HVAC : fbDPT_Switch_pro;
    M2_013_5I202_RT601_CT : fbDPT_Value_Temp_pro;
    M2_014_5I202_RY601_CV : fbDPT_Value_AirQuality_pro;
    M2_015_5I202_LH601_OP : fbDPT_Scaling_pro;
    M2_016_5I202_LH601_CMD : fbDPT_Switch_pro;
    M2_017_5I202_LC601_OP : fbDPT_Scaling_pro;
    M2_018_5I202_LC601_CMD : fbDPT_Switch_pro;
    M2_019_5I202_RT601_SP : fbDPT_Value_Temp_pro;
    M2_020_5I202_RT601_SP_FB : fbDPT_Value_Temp_pro;
    M2_021_5I301_RB601_V : fbDPT_Switch_pro;  (* 5I301 *)
    M2_022_5I301_RB601_HVAC : fbDPT_Switch_pro;
    M2_023_5I301_RT601_CT : fbDPT_Value_Temp_pro;
    M2_024_5I301_RY601_CV : fbDPT_Value_AirQuality_pro;
    M2_025_5I301_LH601_OP : fbDPT_Scaling_pro;
    M2_026_5I301_LH601_CMD : fbDPT_Switch_pro;
    M2_027_5I301_LC601_OP : fbDPT_Scaling_pro;
    M2_028_5I301_LC601_CMD : fbDPT_Switch_pro;
    M2_029_5I301_RT601_SP : fbDPT_Value_Temp_pro;
    M2_030_5I301_RT601_SP_FB : fbDPT_Value_Temp_pro;
    M2_031_5I302_RB601_V : fbDPT_Switch_pro;  (* 5I302 *)
    M2_032_5I302_RB601_HVAC : fbDPT_Switch_pro;
    M2_033_5I302_RT601_CT : fbDPT_Value_Temp_pro;
    M2_034_5I302_RY601_CV : fbDPT_Value_AirQuality_pro;
    M2_035_5I302_LH601_OP : fbDPT_Scaling_pro;
    M2_036_5I302_LH601_CMD : fbDPT_Switch_pro;
    M2_037_5I302_LC601_OP : fbDPT_Scaling_pro;
    M2_038_5I302_LC601_CMD : fbDPT_Switch_pro;
    M2_039_5I302_RT601_SP : fbDPT_Value_Temp_pro;
    M2_040_5I302_RT601_SP_FB : fbDPT_Value_Temp_pro;
    M2_041_5J201_RB601_V : fbDPT_Switch_pro;  (* 5J201 *)
    M2_042_5J201_RB601_HVAC : fbDPT_Switch_pro;
    M2_043_5J201_RT601_CT : fbDPT_Value_Temp_pro;
    M2_044_5J201_RY601_CV : fbDPT_Value_AirQuality_pro;
    M2_045_5J201_LH601_OP : fbDPT_Scaling_pro;
    M2_046_5J201_LH601_CMD : fbDPT_Switch_pro;
    M2_047_5J201_LC601_OP : fbDPT_Scaling_pro;
    M2_048_5J201_LC601_CMD : fbDPT_Switch_pro;
    M2_049_5J201_RT601_SP : fbDPT_Value_Temp_pro;
    M2_050_5J201_RT601_SP_FB : fbDPT_Value_Temp_pro;
    M2_051_5J202_RB601_V : fbDPT_Switch_pro;  (* 5J202 *)
    M2_052_5J202_RB601_HVAC : fbDPT_Switch_pro;
    M2_053_5J202_RT601_CT : fbDPT_Value_Temp_pro;
    M2_054_5J202_RY601_CV : fbDPT_Value_AirQuality_pro;
    M2_055_5J202_LH601_OP : fbDPT_Scaling_pro;
    M2_056_5J202_LH601_CMD : fbDPT_Switch_pro;
    M2_057_5J202_LC601_OP : fbDPT_Scaling_pro;
    M2_058_5J202_LC601_CMD : fbDPT_Switch_pro;
    M2_059_5J202_RT601_SP : fbDPT_Value_Temp_pro;
    M2_060_5J202_RT601_SP_FB : fbDPT_Value_Temp_pro;
    M2_061_5J301_RB601_V : fbDPT_Switch_pro;  (* 5J301 *)
    M2_062_5J301_RB601_HVAC : fbDPT_Switch_pro;
    M2_063_5J301_RT601_CT : fbDPT_Value_Temp_pro;
    M2_064_5J301_RY601_CV : fbDPT_Value_AirQuality_pro;
    M2_065_5J301_LH601_OP : fbDPT_Scaling_pro;
    M2_066_5J301_LH601_CMD : fbDPT_Switch_pro;
    M2_067_5J301_LC601_OP : fbDPT_Scaling_pro;
    M2_068_5J301_LC601_CMD : fbDPT_Switch_pro;
    M2_069_5J301_RT601_SP : fbDPT_Value_Temp_pro;
    M2_070_5J301_RT601_SP_FB : fbDPT_Value_Temp_pro;
    M2_071_5K302_RB601_V : fbDPT_Switch_pro;  (* 5K302 *)
    M2_072_5K302_RB601_HVAC : fbDPT_Switch_pro;
    M2_073_5K302_RT601_CT : fbDPT_Value_Temp_pro;
    M2_074_5K302_RY601_CV : fbDPT_Value_AirQuality_pro;
    M2_075_5K302_LH601_OP : fbDPT_Scaling_pro;
    M2_076_5K302_LH601_CMD : fbDPT_Switch_pro;
    M2_077_5K302_LC601_OP : fbDPT_Scaling_pro;
    M2_078_5K302_LC601_CMD : fbDPT_Switch_pro;
    M2_079_5K302_RT601_SP : fbDPT_Value_Temp_pro;
    M2_080_5K302_RT601_SP_FB : fbDPT_Value_Temp_pro;
    M2_081_5K201_RB601_V : fbDPT_Switch_pro;  (* 5K201 *)
    M2_082_5K201_RB601_HVAC : fbDPT_Switch_pro;
    M2_083_5K201_RT601_CT : fbDPT_Value_Temp_pro;
    M2_084_5K201_RY601_CV : fbDPT_Value_AirQuality_pro;
    M2_085_5K201_LH601_OP : fbDPT_Scaling_pro;
    M2_086_5K201_LH601_CMD : fbDPT_Switch_pro;
    M2_087_5K201_LC601_OP : fbDPT_Scaling_pro;
    M2_088_5K201_LC601_CMD : fbDPT_Switch_pro;
    M2_089_5K201_RT601_SP : fbDPT_Value_Temp_pro;
    M2_090_5K201_RT601_SP_FB : fbDPT_Value_Temp_pro;
    M2_091_5K202_RB601_V : fbDPT_Switch_pro;  (* 5K202 *)
    M2_092_5K202_RB601_HVAC : fbDPT_Switch_pro;
    M2_093_5K202_RT601_CT : fbDPT_Value_Temp_pro;
    M2_094_5K202_RY601_CV : fbDPT_Value_AirQuality_pro;
    M2_095_5K202_LH601_OP : fbDPT_Scaling_pro;
    M2_096_5K202_LH601_CMD : fbDPT_Switch_pro;
    M2_097_5K202_LC601_OP : fbDPT_Scaling_pro;
    M2_098_5K202_LC601_CMD : fbDPT_Switch_pro;
    M2_099_5K202_RT601_SP : fbDPT_Value_Temp_pro;
    M2_100_5K202_RT601_SP_FB : fbDPT_Value_Temp_pro;
    M2_101_5K301_RB601_V : fbDPT_Switch_pro;  (* 5K301 *)
    M2_102_5K301_RB601_HVAC : fbDPT_Switch_pro;
    M2_103_5K301_RT601_CT : fbDPT_Value_Temp_pro;
    M2_104_5K301_RY601_CV : fbDPT_Value_AirQuality_pro;
    M2_105_5K301_LH601_OP : fbDPT_Scaling_pro;
    M2_106_5K301_LH601_CMD : fbDPT_Switch_pro;
    M2_107_5K301_LC601_OP : fbDPT_Scaling_pro;
    M2_108_5K301_LC601_CMD : fbDPT_Switch_pro;
    M2_109_5K301_RT601_SP : fbDPT_Value_Temp_pro;
    M2_110_5K301_RT601_SP_FB : fbDPT_Value_Temp_pro;
    M2_111_5L201_RB601_V : fbDPT_Switch_pro;  (* 5L201 *)
    M2_112_5L201_RB601_HVAC : fbDPT_Switch_pro;
    M2_113_5L201_RT601_CT : fbDPT_Value_Temp_pro;
    M2_114_5L201_RY601_CV : fbDPT_Value_AirQuality_pro;
    M2_115_5L201_LH601_OP : fbDPT_Scaling_pro;
    M2_116_5L201_LH601_CMD : fbDPT_Switch_pro;
    M2_117_5L201_LC601_OP : fbDPT_Scaling_pro;
    M2_118_5L201_LC601_CMD : fbDPT_Switch_pro;
    M2_119_5L201_RT601_SP : fbDPT_Value_Temp_pro;
    M2_120_5L201_RT601_SP_FB : fbDPT_Value_Temp_pro;
    M2_121_5L202_RB601_V : fbDPT_Switch_pro;  (* 5L202 *)
    M2_122_5L202_RB601_HVAC : fbDPT_Switch_pro;
    M2_123_5L202_RT601_CT : fbDPT_Value_Temp_pro;
    M2_124_5L202_RY601_CV : fbDPT_Value_AirQuality_pro;
    M2_125_5L202_LH601_OP : fbDPT_Scaling_pro;
    M2_126_5L202_LH601_CMD : fbDPT_Switch_pro;
    M2_127_5L202_LC601_OP : fbDPT_Scaling_pro;
    M2_128_5L202_LC601_CMD : fbDPT_Switch_pro;
    M2_129_5L202_RT601_SP : fbDPT_Value_Temp_pro;
    M2_130_5L202_RT601_SP_FB : fbDPT_Value_Temp_pro;
    M2_131_5L301_RB601_V : fbDPT_Switch_pro;  (* 5L301 *)
    M2_132_5L301_RB601_HVAC : fbDPT_Switch_pro;
    M2_133_5L301_RT601_CT : fbDPT_Value_Temp_pro;
    M2_134_5L301_RY601_CV : fbDPT_Value_AirQuality_pro;
    M2_135_5L301_LH601_OP : fbDPT_Scaling_pro;
    M2_136_5L301_LH601_CMD : fbDPT_Switch_pro;
    M2_137_5L301_LC601_OP : fbDPT_Scaling_pro;
    M2_138_5L301_LC601_CMD : fbDPT_Switch_pro;
    M2_139_5L301_RT601_SP : fbDPT_Value_Temp_pro;
    M2_140_5L301_RT601_SP_FB : fbDPT_Value_Temp_pro;
    M2_141_5L302_RB601_V : fbDPT_Switch_pro;  (* 5L302 *)
    M2_142_5L302_RB601_HVAC : fbDPT_Switch_pro;
    M2_143_5L302_RT601_CT : fbDPT_Value_Temp_pro;
    M2_144_5L302_RY601_CV : fbDPT_Value_AirQuality_pro;
    M2_145_5L302_LH601_OP : fbDPT_Scaling_pro;
    M2_146_5L302_LH601_CMD : fbDPT_Switch_pro;
    M2_147_5L302_LC601_OP : fbDPT_Scaling_pro;
    M2_148_5L302_LC601_CMD : fbDPT_Switch_pro;
    M2_149_5L302_RT601_SP : fbDPT_Value_Temp_pro;
    M2_150_5L302_RT601_SP_FB : fbDPT_Value_Temp_pro;
    M2_151_5M201_RB601_V : fbDPT_Switch_pro;  (* 5M201 *)
    M2_152_5M201_RB601_HVAC : fbDPT_Switch_pro;
    M2_153_5M201_RT601_CT : fbDPT_Value_Temp_pro;
    M2_154_5M201_RY601_CV : fbDPT_Value_AirQuality_pro;
    M2_155_5M201_LH601_OP : fbDPT_Scaling_pro;
    M2_156_5M201_LH601_CMD : fbDPT_Switch_pro;
    M2_157_5M201_LC601_OP : fbDPT_Scaling_pro;
    M2_158_5M201_LC601_CMD : fbDPT_Switch_pro;
    M2_159_5M201_RT601_SP : fbDPT_Value_Temp_pro;
    M2_160_5M201_RT601_SP_FB : fbDPT_Value_Temp_pro;
    M2_161_5M202_RB601_V : fbDPT_Switch_pro;  (* 5M202 *)
    M2_162_5M202_RB601_HVAC : fbDPT_Switch_pro;
    M2_163_5M202_RT601_CT : fbDPT_Value_Temp_pro;
    M2_164_5M202_RY601_CV : fbDPT_Value_AirQuality_pro;
    M2_165_5M202_LH601_OP : fbDPT_Scaling_pro;
    M2_166_5M202_LH601_CMD : fbDPT_Switch_pro;
    M2_167_5M202_LC601_OP : fbDPT_Scaling_pro;
    M2_168_5M202_LC601_CMD : fbDPT_Switch_pro;
    M2_169_5M202_RT601_SP : fbDPT_Value_Temp_pro;
    M2_170_5M202_RT601_SP_FB : fbDPT_Value_Temp_pro;
    M2_171_5M301_RB601_V : fbDPT_Switch_pro;  (* 5M301 *)
    M2_172_5M301_RB601_HVAC : fbDPT_Switch_pro;
    M2_173_5M301_RT601_CT : fbDPT_Value_Temp_pro;
    M2_174_5M301_RY601_CV : fbDPT_Value_AirQuality_pro;
    M2_175_5M301_LH601_OP : fbDPT_Scaling_pro;
    M2_176_5M301_LH601_CMD : fbDPT_Switch_pro;
    M2_177_5M301_LC601_OP : fbDPT_Scaling_pro;
    M2_178_5M301_LC601_CMD : fbDPT_Switch_pro;
    M2_179_5M301_RT601_SP : fbDPT_Value_Temp_pro;
    M2_180_5M301_RT601_SP_FB : fbDPT_Value_Temp_pro;
    M2_181_5N201_RB601_V : fbDPT_Switch_pro;  (* 5N201 *)
    M2_182_5N201_RB601_HVAC : fbDPT_Switch_pro;
    M2_183_5N201_RT601_CT : fbDPT_Value_Temp_pro;
    M2_184_5N201_RY601_CV : fbDPT_Value_AirQuality_pro;
    M2_185_5N201_LH601_OP : fbDPT_Scaling_pro;
    M2_186_5N201_LH601_CMD : fbDPT_Switch_pro;
    M2_187_5N201_LC601_OP : fbDPT_Scaling_pro;
    M2_188_5N201_LC601_CMD : fbDPT_Switch_pro;
    M2_189_5N201_RT601_SP : fbDPT_Value_Temp_pro;
    M2_190_5N201_RT601_SP_FB : fbDPT_Value_Temp_pro;
    M2_191_5N202_RB601_V : fbDPT_Switch_pro;  (* 5N202 *)
    M2_192_5N202_RB601_HVAC : fbDPT_Switch_pro;
    M2_193_5N202_RT601_CT : fbDPT_Value_Temp_pro;
    M2_194_5N202_RY601_CV : fbDPT_Value_AirQuality_pro;
    M2_195_5N202_LH601_OP : fbDPT_Scaling_pro;
    M2_196_5N202_LH601_CMD : fbDPT_Switch_pro;
    M2_197_5N202_LC601_OP : fbDPT_Scaling_pro;
    M2_198_5N202_LC601_CMD : fbDPT_Switch_pro;
    M2_199_5N202_RT601_SP : fbDPT_Value_Temp_pro;
    M2_200_5N202_RT601_SP_FB : fbDPT_Value_Temp_pro;
    M2_201_5N301_RB601_V : fbDPT_Switch_pro;  (* 5N301 *)
    M2_202_5N301_RB601_HVAC : fbDPT_Switch_pro;
    M2_203_5N301_RT601_CT : fbDPT_Value_Temp_pro;
    M2_204_5N301_RY601_CV : fbDPT_Value_AirQuality_pro;
    M2_205_5N301_LH601_OP : fbDPT_Scaling_pro;
    M2_206_5N301_LH601_CMD : fbDPT_Switch_pro;
    M2_207_5N301_LC601_OP : fbDPT_Scaling_pro;
    M2_208_5N301_LC601_CMD : fbDPT_Switch_pro;
    M2_209_5N301_RT601_SP : fbDPT_Value_Temp_pro;
    M2_210_5N301_RT601_SP_FB : fbDPT_Value_Temp_pro;
    M2_211_5N302_RB601_V : fbDPT_Switch_pro;  (* 5N302 *)
    M2_212_5N302_RB601_HVAC : fbDPT_Switch_pro;
    M2_213_5N302_RT601_CT : fbDPT_Value_Temp_pro;
    M2_214_5N302_RY601_CV : fbDPT_Value_AirQuality_pro;
    M2_215_5N302_LH601_OP : fbDPT_Scaling_pro;
    M2_216_5N302_LH601_CMD : fbDPT_Switch_pro;
    M2_217_5N302_LC601_OP : fbDPT_Scaling_pro;
    M2_218_5N302_LC601_CMD : fbDPT_Switch_pro;
    M2_219_5N302_RT601_SP : fbDPT_Value_Temp_pro;
    M2_220_5N302_RT601_SP_FB : fbDPT_Value_Temp_pro;
    M2_221_5O302_RB601_V : fbDPT_Switch_pro;  (* 5O302 *)
    M2_222_5O302_RB601_HVAC : fbDPT_Switch_pro;
    M2_223_5O302_RT601_CT : fbDPT_Value_Temp_pro;
    M2_224_5O302_RY601_CV : fbDPT_Value_AirQuality_pro;
    M2_225_5O302_LH601_OP : fbDPT_Scaling_pro;
    M2_226_5O302_LH601_CMD : fbDPT_Switch_pro;
    M2_227_5O302_LC601_OP : fbDPT_Scaling_pro;
    M2_228_5O302_LC601_CMD : fbDPT_Switch_pro;
    M2_229_5O302_RT601_SP : fbDPT_Value_Temp_pro;
    M2_230_5O302_RT601_SP_FB : fbDPT_Value_Temp_pro;
    M2_231_5O201_RB601_V : fbDPT_Switch_pro;  (* 5O201 *)
    M2_232_5O201_RB601_HVAC : fbDPT_Switch_pro;
    M2_233_5O201_RT601_CT : fbDPT_Value_Temp_pro;
    M2_234_5O201_RY601_CV : fbDPT_Value_AirQuality_pro;
    M2_235_5O201_LH601_OP : fbDPT_Scaling_pro;
    M2_236_5O201_LH601_CMD : fbDPT_Switch_pro;
    M2_237_5O201_LC601_OP : fbDPT_Scaling_pro;
    M2_238_5O201_LC601_CMD : fbDPT_Switch_pro;
    M2_239_5O201_RT601_SP : fbDPT_Value_Temp_pro;
    M2_240_5O201_RT601_SP_FB : fbDPT_Value_Temp_pro;
    M2_241_5O202_RB601_V : fbDPT_Switch_pro;  (* 5O202 *)
    M2_242_5O202_RB601_HVAC : fbDPT_Switch_pro;
    M2_243_5O202_RT601_CT : fbDPT_Value_Temp_pro;
    M2_244_5O202_RY601_CV : fbDPT_Value_AirQuality_pro;
    M2_245_5O202_LH601_OP : fbDPT_Scaling_pro;
    M2_246_5O202_LH601_CMD : fbDPT_Switch_pro;
    M2_247_5O202_LC601_OP : fbDPT_Scaling_pro;
    M2_248_5O202_LC601_CMD : fbDPT_Switch_pro;
    M2_249_5O202_RT601_SP : fbDPT_Value_Temp_pro;
    M2_250_5O202_RT601_SP_FB : fbDPT_Value_Temp_pro;
  END_VAR

